LIN {X 0,Y 366.055,Z 486.683,A -85,B 0,C 180,E1 -21663.434,E2 -21663.434} C_VEL
LIN {X 0,Y 364.924,Z 500.957,A -85,B 0,C 180,E1 -21663.921,E2 -21663.921} C_VEL
LIN {X 0,Y 363.137,Z 514.776,A -85,B 0,C 180,E1 -21664.588,E2 -21664.588} C_VEL
LIN {X 0,Y 361.174,Z 526.804,A -85,B 0,C 180,E1 -21665.361,E2 -21665.361} C_VEL
LIN {X 0,Y 358.835,Z 539.501,A -85,B 0,C 180,E1 -21666.415,E2 -21666.415} C_VEL
LIN {X 0,Y 356.342,Z 551.532,A -85,B 0,C 180,E1 -21667.677,E2 -21667.677} C_VEL
LIN {X 0,Y 353.739,Z 562.686,A -85,B 0,C 180,E1 -21669.123,E2 -21669.123} C_VEL
LIN {X 0,Y 351.083,Z 573.104,A -85,B 0,C 180,E1 -21670.784,E2 -21670.784} C_VEL
LIN {X 0,Y 348.812,Z 581.735,A -85,B 0,C 180,E1 -21672.473,E2 -21672.473} C_VEL
LIN {X 0,Y 346.741,Z 590.061,A -85,B 0,C 180,E1 -21674.478,E2 -21674.478} C_VEL
LIN {X 0,Y 345.082,Z 596.796,A -85,B 0,C 180,E1 -21676.504,E2 -21676.504} C_VEL
LIN {X 0,Y 343.677,Z 602.83,A -85,B 0,C 180,E1 -21678.839,E2 -21678.839} C_VEL
LIN {X 0,Y 342.95,Z 606.345,A -85,B 0,C 180,E1 -21680.599,E2 -21680.599} C_VEL
LIN {X 0,Y 342.378,Z 609.772,A -85,B 0,C 180,E1 -21682.952,E2 -21682.952} C_VEL
LIN {X 0,Y 342.438,Z 612.217,A -85,B 0,C 180,E1 -21685.604,E2 -21685.604} C_VEL
LIN {X 0,Y 342.403,Z 616.736,A -85,B 0,C 180,E1 -21687.658,E2 -21687.658} C_VEL
LIN {X 0,Y 342.425,Z 618.738,A -85,B 0,C 180,E1 -21688.831,E2 -21688.831} C_VEL
LIN {X 0,Y 342.348,Z 621.565,A -85,B 0,C 180,E1 -21691.175,E2 -21691.175} C_VEL
LIN {X 0,Y 342.211,Z 622.906,A -85,B 0,C 180,E1 -21693.523,E2 -21693.523} C_VEL
LIN {X 0,Y 342.409,Z 622.824,A -85,B 0,C 180,E1 -21695.873,E2 -21695.873} C_VEL
LIN {X 0,Y 342.854,Z 621.327,A -85,B 0,C 180,E1 -21698.225,E2 -21698.225} C_VEL
LIN {X 0,Y 344.003,Z 618.414,A -85,B 0,C 180,E1 -21700.562,E2 -21700.562} C_VEL
LIN {X 0,Y 345.62,Z 614.037,A -85,B 0,C 180,E1 -21702.884,E2 -21702.884} C_VEL
LIN {X 0,Y 347.136,Z 609.753,A -85,B 0,C 180,E1 -21704.612,E2 -21704.612} C_VEL
LIN {X 0,Y 349.775,Z 602.476,A -85,B 0,C 180,E1 -21706.883,E2 -21706.883} C_VEL
LIN {X 0,Y 352.529,Z 594.517,A -85,B 0,C 180,E1 -21708.839,E2 -21708.839} C_VEL
LIN {X 0,Y 355.143,Z 586.331,A -85,B 0,C 180,E1 -21710.495,E2 -21710.495} C_VEL
LIN {X 0,Y 358.31,Z 576.517,A -85,B 0,C 180,E1 -21712.108,E2 -21712.108} C_VEL
LIN {X 0,Y 361.68,Z 564.796,A -85,B 0,C 180,E1 -21713.697,E2 -21713.697} C_VEL
LIN {X 0,Y 364.915,Z 552.862,A -85,B 0,C 180,E1 -21714.981,E2 -21714.981} C_VEL
LIN {X 0,Y 367.967,Z 539.899,A -85,B 0,C 180,E1 -21716.119,E2 -21716.119} C_VEL
LIN {X 0,Y 370.614,Z 527.481,A -85,B 0,C 180,E1 -21716.977,E2 -21716.977} C_VEL
LIN {X 0,Y 372.935,Z 514.221,A -85,B 0,C 180,E1 -21717.703,E2 -21717.703} C_VEL
LIN {X 0,Y 375.156,Z 498.538,A -85,B 0,C 180,E1 -21718.326,E2 -21718.326} C_VEL
LIN {X 0,Y 383.083,Z 416.624,A -85,B 0,C 180,E1 -21720.797,E2 -21720.797} C_VEL
LIN {X 0,Y 382.44,Z 396.943,A -85,B 0,C 180,E1 -21721.901,E2 -21721.901} C_VEL
LIN {X 0,Y 380.969,Z 378.673,A -85,B 0,C 180,E1 -21723.164,E2 -21723.164} C_VEL
LIN {X 0,Y 380.508,Z 375.676,A -85,B 0,C 180,E1 -21723.428,E2 -21723.428} C_VEL
LIN {X 0,Y 378.135,Z 368.085,A -85,B 0,C 180,E1 -21724.4,E2 -21724.4} C_VEL
LIN {X 0,Y 372.813,Z 359.888,A -85,B 0,C 180,E1 -21726.277,E2 -21726.277} C_VEL
LIN {X 0,Y 367.268,Z 352.213,A -85,B 0,C 180,E1 -21728.561,E2 -21728.561} C_VEL
LIN {X 0,Y 364.472,Z 347.395,A -85,B 0,C 180,E1 -21730.802,E2 -21730.802} C_VEL
LIN {X 0,Y 362.586,Z 344.058,A -85,B 0,C 180,E1 -21732.77,E2 -21732.77} C_VEL
LIN {X 0,Y 360.384,Z 340.995,A -85,B 0,C 180,E1 -21735.597,E2 -21735.597} C_VEL
LIN {X 0,Y 359.374,Z 339.035,A -85,B 0,C 180,E1 -21738.495,E2 -21738.495} C_VEL
LIN {X 0,Y 359.081,Z 338.68,A -85,B 0,C 180,E1 -21739.93,E2 -21739.93} C_VEL
LIN {X 0,Y 358.94,Z 338.821,A -85,B 0,C 180,E1 -21741.358,E2 -21741.358} C_VEL
LIN {X 0,Y 359.063,Z 340.127,A -85,B 0,C 180,E1 -21744.181,E2 -21744.181} C_VEL
LIN {X 0,Y 359.917,Z 342.545,A -85,B 0,C 180,E1 -21746.981,E2 -21746.981} C_VEL
LIN {X 0,Y 361.292,Z 346.17,A -85,B 0,C 180,E1 -21749.73,E2 -21749.73} C_VEL
LIN {X 0,Y 362.561,Z 349.811,A -85,B 0,C 180,E1 -21751.77,E2 -21751.77} C_VEL
LIN {X 0,Y 367.024,Z 356.698,A -85,B 0,C 180,E1 -21754.033,E2 -21754.033} C_VEL
LIN {X 0,Y 370.271,Z 361.948,A -85,B 0,C 180,E1 -21755.437,E2 -21755.437} C_VEL
LIN {X 0,Y 373.65,Z 367.876,A -85,B 0,C 180,E1 -21756.763,E2 -21756.763} C_VEL
LIN {X 0,Y 377.509,Z 375.052,A -85,B 0,C 180,E1 -21758.145,E2 -21758.145} C_VEL
LIN {X 0,Y 382.443,Z 385.972,A -85,B 0,C 180,E1 -21759.817,E2 -21759.817} C_VEL
LIN {X 0,Y 383.625,Z 389.184,A -85,B 0,C 180,E1 -21760.215,E2 -21760.215} C_VEL
LIN {X 0,Y 384.825,Z 399.873,A -85,B 0,C 180,E1 -21760.981,E2 -21760.981} C_VEL
LIN {X 0,Y 375.817,Z 490.766,A -85,B 0,C 180,E1 -21763.696,E2 -21763.696} C_VEL
LIN {X 0,Y 373.695,Z 505.863,A -85,B 0,C 180,E1 -21764.369,E2 -21764.369} C_VEL
LIN {X 0,Y 371.24,Z 520.286,A -85,B 0,C 180,E1 -21765.243,E2 -21765.243} C_VEL
LIN {X 0,Y 368.417,Z 533.693,A -85,B 0,C 180,E1 -21766.276,E2 -21766.276} C_VEL
LIN {X 0,Y 365.648,Z 545.087,A -85,B 0,C 180,E1 -21767.372,E2 -21767.372} C_VEL
LIN {X 0,Y 362.523,Z 556.587,A -85,B 0,C 180,E1 -21768.718,E2 -21768.718} C_VEL
LIN {X 0,Y 359.5,Z 566.8,A -85,B 0,C 180,E1 -21770.184,E2 -21770.184} C_VEL
LIN {X 0,Y 356.513,Z 576.165,A -85,B 0,C 180,E1 -21771.811,E2 -21771.811} C_VEL
LIN {X 0,Y 353.399,Z 585.186,A -85,B 0,C 180,E1 -21773.742,E2 -21773.742} C_VEL
LIN {X 0,Y 350.892,Z 591.603,A -85,B 0,C 180,E1 -21775.42,E2 -21775.42} C_VEL
LIN {X 0,Y 348.777,Z 596.889,A -85,B 0,C 180,E1 -21777.122,E2 -21777.122} C_VEL
LIN {X 0,Y 346.492,Z 602.436,A -85,B 0,C 180,E1 -21779.421,E2 -21779.421} C_VEL
LIN {X 0,Y 345.156,Z 605.533,A -85,B 0,C 180,E1 -21781.163,E2 -21781.163} C_VEL
LIN {X 0,Y 343.894,Z 608.425,A -85,B 0,C 180,E1 -21783.563,E2 -21783.563} C_VEL
LIN {X 0,Y 342.925,Z 609.815,A -85,B 0,C 180,E1 -21785.862,E2 -21785.862} C_VEL
LIN {X 0,Y 342.295,Z 609.846,A -85,B 0,C 180,E1 -21788.235,E2 -21788.235} C_VEL
LIN {X 0,Y 342.083,Z 608.426,A -85,B 0,C 180,E1 -21790.619,E2 -21790.619} C_VEL
LIN {X 0,Y 341.946,Z 605.459,A -85,B 0,C 180,E1 -21793.022,E2 -21793.022} C_VEL
LIN {X 0,Y 342.078,Z 602.213,A -85,B 0,C 180,E1 -21794.83,E2 -21794.83} C_VEL
LIN {X 0,Y 342.277,Z 597.919,A -85,B 0,C 180,E1 -21796.648,E2 -21796.648} C_VEL
LIN {X 0,Y 342.562,Z 591.515,A -85,B 0,C 180,E1 -21798.787,E2 -21798.787} C_VEL
LIN {X 0,Y 343.068,Z 583.313,A -85,B 0,C 180,E1 -21800.934,E2 -21800.934} C_VEL
LIN {X 0,Y 343.699,Z 573.569,A -85,B 0,C 180,E1 -21802.983,E2 -21802.983} C_VEL
LIN {X 0,Y 344.435,Z 563.987,A -85,B 0,C 180,E1 -21804.638,E2 -21804.638} C_VEL
LIN {X 0,Y 345.258,Z 553.252,A -85,B 0,C 180,E1 -21806.184,E2 -21806.184} C_VEL
LIN {X 0,Y 346.21,Z 541.181,A -85,B 0,C 180,E1 -21807.613,E2 -21807.613} C_VEL
LIN {X 0,Y 347.26,Z 527.207,A -85,B 0,C 180,E1 -21808.953,E2 -21808.953} C_VEL
LIN {X 0,Y 348.192,Z 513.062,A -85,B 0,C 180,E1 -21810.026,E2 -21810.026} C_VEL
LIN {X 0,Y 349.048,Z 498.453,A -85,B 0,C 180,E1 -21810.862,E2 -21810.862} C_VEL
LIN {X 0,Y 349.81,Z 482.818,A -85,B 0,C 180,E1 -21811.499,E2 -21811.499} C_VEL
LIN {X 0,Y 353.103,Z 383.38,A -85,B 0,C 180,E1 -21814.323,E2 -21814.323} C_VEL
LIN {X 0,Y 349.382,Z 350.073,A -85,B 0,C 180,E1 -21815.44,E2 -21815.44} C_VEL
LIN {X 0,Y 349.055,Z 345.645,A -85,B 0,C 180,E1 -21815.587,E2 -21815.587} C_VEL
LIN {X 0,Y 349.57,Z 337.879,A -85,B 0,C 180,E1 -21816.95,E2 -21816.95} C_VEL
LIN {X 0,Y 346.602,Z 322.549,A -85,B 0,C 180,E1 -21819.828,E2 -21819.828} C_VEL
LIN {X 0,Y 344.862,Z 314.085,A -85,B 0,C 180,E1 -21821.46,E2 -21821.46} C_VEL
LIN {X 0,Y 344.806,Z 314.085,A -85,B 0,C 180,E1 -21825.316,E2 -21825.316} C_VEL
LIN {X 0,Y 344.819,Z 314.088,A -85,B 0,C 180,E1 -21828.729,E2 -21828.729} C_VEL
LIN {X 0,Y 344.839,Z 314.089,A -85,B 0,C 180,E1 -21832.454,E2 -21832.454} C_VEL
LIN {X 0,Y 344.839,Z 314.08,A -85,B 0,C 180,E1 -21836.388,E2 -21836.388} C_VEL
LIN {X 0,Y 344.826,Z 314.088,A -85,B 0,C 180,E1 -21839.478,E2 -21839.478} C_VEL
LIN {X 0,Y 344.883,Z 314.078,A -85,B 0,C 180,E1 -21843.458,E2 -21843.458} C_VEL
LIN {X 0,Y 344.895,Z 314.079,A -85,B 0,C 180,E1 -21847.3,E2 -21847.3} C_VEL
LIN {X 0,Y 344.938,Z 314.077,A -85,B 0,C 180,E1 -21849.803,E2 -21849.803} C_VEL
LIN {X 0,Y 344.982,Z 314.067,A -85,B 0,C 180,E1 -21853.483,E2 -21853.483} C_VEL
LIN {X 0,Y 345.054,Z 314.156,A -85,B 0,C 180,E1 -21856.537,E2 -21856.537} C_VEL
LIN {X 0,Y 346.568,Z 318.213,A -85,B 0,C 180,E1 -21856.725,E2 -21856.725} C_VEL
LIN {X 0,Y 351.173,Z 329.859,A -85,B 0,C 180,E1 -21857.271,E2 -21857.271} C_VEL
LIN {X 0,Y 356.843,Z 346.888,A -85,B 0,C 180,E1 -21857.977,E2 -21857.977} C_VEL
LIN {X 0,Y 354.437,Z 447.995,A -85,B 0,C 180,E1 -21860.004,E2 -21860.004} C_VEL
LIN {X 0,Y 353.812,Z 462.506,A -85,B 0,C 180,E1 -21860.526,E2 -21860.526} C_VEL
LIN {X 0,Y 352.973,Z 476.914,A -85,B 0,C 180,E1 -21861.294,E2 -21861.294} C_VEL
LIN {X 0,Y 351.93,Z 488.862,A -85,B 0,C 180,E1 -21862.133,E2 -21862.133} C_VEL
LIN {X 0,Y 350.837,Z 500.065,A -85,B 0,C 180,E1 -21863.117,E2 -21863.117} C_VEL
LIN {X 0,Y 349.324,Z 511.865,A -85,B 0,C 180,E1 -21864.388,E2 -21864.388} C_VEL
LIN {X 0,Y 348.282,Z 521.61,A -85,B 0,C 180,E1 -21865.672,E2 -21865.672} C_VEL
LIN {X 0,Y 347.134,Z 530.782,A -85,B 0,C 180,E1 -21867.106,E2 -21867.106} C_VEL
LIN {X 0,Y 345.831,Z 539.993,A -85,B 0,C 180,E1 -21868.837,E2 -21868.837} C_VEL
LIN {X 0,Y 344.833,Z 547.662,A -85,B 0,C 180,E1 -21870.579,E2 -21870.579} C_VEL
LIN {X 0,Y 344.135,Z 554.022,A -85,B 0,C 180,E1 -21872.33,E2 -21872.33} C_VEL
LIN {X 0,Y 343.661,Z 559.279,A -85,B 0,C 180,E1 -21874.088,E2 -21874.088} C_VEL
LIN {X 0,Y 342.988,Z 564.867,A -85,B 0,C 180,E1 -21876.446,E2 -21876.446} C_VEL
LIN {X 0,Y 342.651,Z 568.004,A -85,B 0,C 180,E1 -21878.224,E2 -21878.224} C_VEL
LIN {X 0,Y 342.579,Z 570.938,A -85,B 0,C 180,E1 -21880.601,E2 -21880.601} C_VEL
LIN {X 0,Y 342.606,Z 572.515,A -85,B 0,C 180,E1 -21882.993,E2 -21882.993} C_VEL
LIN {X 0,Y 342.927,Z 572.738,A -85,B 0,C 180,E1 -21885.395,E2 -21885.395} C_VEL
LIN {X 0,Y 343.503,Z 571.602,A -85,B 0,C 180,E1 -21887.807,E2 -21887.807} C_VEL
LIN {X 0,Y 344.465,Z 569.036,A -85,B 0,C 180,E1 -21890.22,E2 -21890.22} C_VEL
LIN {X 0,Y 345.851,Z 564.953,A -85,B 0,C 180,E1 -21892.628,E2 -21892.628} C_VEL
LIN {X 0,Y 347.611,Z 559.233,A -85,B 0,C 180,E1 -21895.03,E2 -21895.03} C_VEL
LIN {X 0,Y 349.574,Z 552.707,A -85,B 0,C 180,E1 -21897.116,E2 -21897.116} C_VEL
LIN {X 0,Y 351.883,Z 544.776,A -85,B 0,C 180,E1 -21899.12,E2 -21899.12} C_VEL
LIN {X 0,Y 354.236,Z 535.872,A -85,B 0,C 180,E1 -21900.934,E2 -21900.934} C_VEL
LIN {X 0,Y 356.818,Z 525.291,A -85,B 0,C 180,E1 -21902.668,E2 -21902.668} C_VEL
LIN {X 0,Y 359.163,Z 514.547,A -85,B 0,C 180,E1 -21904.099,E2 -21904.099} C_VEL
LIN {X 0,Y 361.532,Z 502.269,A -85,B 0,C 180,E1 -21905.42,E2 -21905.42} C_VEL
LIN {X 0,Y 363.519,Z 489.69,A -85,B 0,C 180,E1 -21906.502,E2 -21906.502} C_VEL
LIN {X 0,Y 365.141,Z 475.959,A -85,B 0,C 180,E1 -21907.431,E2 -21907.431} C_VEL
LIN {X 0,Y 366.527,Z 461.755,A -85,B 0,C 180,E1 -21908.123,E2 -21908.123} C_VEL
LIN {X 0,Y 367.394,Z 447.635,A -85,B 0,C 180,E1 -21908.586,E2 -21908.586} C_VEL
LIN {X 0,Y 370.195,Z 363.744,A -85,B 0,C 180,E1 -21910.241,E2 -21910.241} C_VEL
LIN {X 0,Y 361.979,Z 345.819,A -85,B 0,C 180,E1 -21911.518,E2 -21911.518} C_VEL
LIN {X 0,Y 353.326,Z 329.446,A -85,B 0,C 180,E1 -21912.891,E2 -21912.891} C_VEL
LIN {X 0,Y 346.517,Z 317.849,A -85,B 0,C 180,E1 -21914.006,E2 -21914.006} C_VEL
LIN {X 0,Y 345.037,Z 315.104,A -85,B 0,C 180,E1 -21914.262,E2 -21914.262} C_VEL
LIN {X 0,Y 344.79,Z 314.078,A -85,B 0,C 180,E1 -21914.566,E2 -21914.566} C_VEL
LIN {X 0,Y 344.782,Z 314.085,A -85,B 0,C 180,E1 -21916.034,E2 -21916.034} C_VEL
LIN {X 0,Y 344.132,Z 314.178,A -85,B 0,C 180,E1 -21917.008,E2 -21917.008} C_VEL
LIN {X 0,Y 341.252,Z 314.534,A -85,B 0,C 180,E1 -21918.591,E2 -21918.591} C_VEL
LIN {X 0,Y 338.818,Z 314.835,A -85,B 0,C 180,E1 -21919.874,E2 -21919.874} C_VEL
LIN {X 0,Y 337.804,Z 314.962,A -85,B 0,C 180,E1 -21920.867,E2 -21920.867} C_VEL
LIN {X 0,Y 337.739,Z 314.971,A -85,B 0,C 180,E1 -21921.203,E2 -21921.203} C_VEL
LIN {X 0,Y 337.782,Z 314.932,A -85,B 0,C 180,E1 -21924.506,E2 -21924.506} C_VEL
LIN {X 0,Y 337.796,Z 314.961,A -85,B 0,C 180,E1 -21928.223,E2 -21928.223} C_VEL
LIN {X 0,Y 337.823,Z 314.959,A -85,B 0,C 180,E1 -21931.518,E2 -21931.518} C_VEL
LIN {X 0,Y 337.82,Z 314.957,A -85,B 0,C 180,E1 -21935.501,E2 -21935.501} C_VEL
LIN {X 0,Y 337.877,Z 314.955,A -85,B 0,C 180,E1 -21939.364,E2 -21939.364} C_VEL
LIN {X 0,Y 337.892,Z 314.952,A -85,B 0,C 180,E1 -21943.129,E2 -21943.129} C_VEL
LIN {X 0,Y 338.007,Z 314.927,A -85,B 0,C 180,E1 -21946.882,E2 -21946.882} C_VEL
LIN {X 0,Y 338.028,Z 314.921,A -85,B 0,C 180,E1 -21950.458,E2 -21950.458} C_VEL
LIN {X 0,Y 338.186,Z 314.916,A -85,B 0,C 180,E1 -21954.056,E2 -21954.056} C_VEL
LIN {X 0,Y 338.218,Z 314.902,A -85,B 0,C 180,E1 -21957.626,E2 -21957.626} C_VEL
LIN {X 0,Y 338.191,Z 314.898,A -85,B 0,C 180,E1 -21961.187,E2 -21961.187} C_VEL
LIN {X 0,Y 338.226,Z 314.913,A -85,B 0,C 180,E1 -21964.752,E2 -21964.752} C_VEL
LIN {X 0,Y 338.075,Z 314.915,A -85,B 0,C 180,E1 -21968.339,E2 -21968.339} C_VEL
LIN {X 0,Y 338.021,Z 314.919,A -85,B 0,C 180,E1 -21971.959,E2 -21971.959} C_VEL
LIN {X 0,Y 337.911,Z 314.945,A -85,B 0,C 180,E1 -21975.633,E2 -21975.633} C_VEL
LIN {X 0,Y 337.863,Z 314.939,A -85,B 0,C 180,E1 -21978.118,E2 -21978.118} C_VEL
LIN {X 0,Y 337.863,Z 314.947,A -85,B 0,C 180,E1 -21981.115,E2 -21981.115} C_VEL
LIN {X 0,Y 337.82,Z 314.964,A -85,B 0,C 180,E1 -21984.5,E2 -21984.5} C_VEL
LIN {X 0,Y 337.823,Z 314.964,A -85,B 0,C 180,E1 -21988.482,E2 -21988.482} C_VEL
LIN {X 0,Y 337.801,Z 314.962,A -85,B 0,C 180,E1 -21991.779,E2 -21991.779} C_VEL
LIN {X 0,Y 337.829,Z 314.92,A -85,B 0,C 180,E1 -21995.489,E2 -21995.489} C_VEL
LIN {X 0,Y 337.832,Z 314.959,A -85,B 0,C 180,E1 -21998.463,E2 -21998.463} C_VEL
LIN {X 0,Y 337.803,Z 314.966,A -85,B 0,C 180,E1 -22001.72,E2 -22001.72} C_VEL
LIN {X 0,Y 337.796,Z 314.96,A -85,B 0,C 180,E1 -22005.174,E2 -22005.174} C_VEL
LIN {X 0,Y 337.835,Z 314.994,A -85,B 0,C 180,E1 -22008.144,E2 -22008.144} C_VEL
LIN {X 0,Y 341.432,Z 327.545,A -85,B 0,C 180,E1 -22012.321,E2 -22012.321} C_VEL
LIN {X 0,Y 344.132,Z 338.395,A -85,B 0,C 180,E1 -22015.595,E2 -22015.595} C_VEL
LIN {X 0,Y 345.966,Z 346.803,A -85,B 0,C 180,E1 -22017.913,E2 -22017.913} C_VEL
LIN {X 0,Y 354.721,Z 365.775,A -85,B 0,C 180,E1 -22019.409,E2 -22019.409} C_VEL
LIN {X 0,Y 360.3,Z 397.531,A -85,B 0,C 180,E1 -22020.776,E2 -22020.776} C_VEL
LIN {X 0,Y 362.564,Z 414.669,A -85,B 0,C 180,E1 -22021.409,E2 -22021.409} C_VEL
LIN {X 0,Y 360.53,Z 473.255,A -85,B 0,C 180,E1 -22022.564,E2 -22022.564} C_VEL
LIN {X 0,Y 359.715,Z 490.214,A -85,B 0,C 180,E1 -22022.967,E2 -22022.967} C_VEL
LIN {X 0,Y 358.306,Z 504.713,A -85,B 0,C 180,E1 -22023.519,E2 -22023.519} C_VEL
LIN {X 0,Y 356.373,Z 518.008,A -85,B 0,C 180,E1 -22024.227,E2 -22024.227} C_VEL
LIN {X 0,Y 354.175,Z 530.938,A -85,B 0,C 180,E1 -22025.153,E2 -22025.153} C_VEL
LIN {X 0,Y 351.494,Z 544.041,A -85,B 0,C 180,E1 -22026.36,E2 -22026.36} C_VEL
LIN {X 0,Y 348.884,Z 555.826,A -85,B 0,C 180,E1 -22027.735,E2 -22027.735} C_VEL
LIN {X 0,Y 346.211,Z 566.513,A -85,B 0,C 180,E1 -22029.268,E2 -22029.268} C_VEL
LIN {X 0,Y 343.558,Z 576.181,A -85,B 0,C 180,E1 -22030.965,E2 -22030.965} C_VEL
LIN {X 0,Y 341.389,Z 584.236,A -85,B 0,C 180,E1 -22032.696,E2 -22032.696} C_VEL
LIN {X 0,Y 339.34,Z 591.996,A -85,B 0,C 180,E1 -22034.745,E2 -22034.745} C_VEL
LIN {X 0,Y 337.72,Z 598.264,A -85,B 0,C 180,E1 -22036.815,E2 -22036.815} C_VEL
LIN {X 0,Y 336.364,Z 603.864,A -85,B 0,C 180,E1 -22039.201,E2 -22039.201} C_VEL
LIN {X 0,Y 335.534,Z 607.949,A -85,B 0,C 180,E1 -22041.6,E2 -22041.6} C_VEL
LIN {X 0,Y 335.275,Z 610.63,A -85,B 0,C 180,E1 -22044.007,E2 -22044.007} C_VEL
LIN {X 0,Y 335.369,Z 611.745,A -85,B 0,C 180,E1 -22045.661,E2 -22045.661} C_VEL
LIN {X 0,Y 335.337,Z 616.072,A -85,B 0,C 180,E1 -22047.609,E2 -22047.609} C_VEL
LIN {X 0,Y 335.361,Z 618.154,A -85,B 0,C 180,E1 -22048.806,E2 -22048.806} C_VEL
LIN {X 0,Y 335.259,Z 621.129,A -85,B 0,C 180,E1 -22051.2,E2 -22051.2} C_VEL
LIN {X 0,Y 335.135,Z 622.628,A -85,B 0,C 180,E1 -22053.598,E2 -22053.598} C_VEL
LIN {X 0,Y 335.333,Z 622.712,A -85,B 0,C 180,E1 -22055.998,E2 -22055.998} C_VEL
LIN {X 0,Y 335.815,Z 621.404,A -85,B 0,C 180,E1 -22058.398,E2 -22058.398} C_VEL
LIN {X 0,Y 337.027,Z 618.708,A -85,B 0,C 180,E1 -22060.783,E2 -22060.783} C_VEL
LIN {X 0,Y 338.709,Z 614.527,A -85,B 0,C 180,E1 -22063.151,E2 -22063.151} C_VEL
LIN {X 0,Y 340.3,Z 610.395,A -85,B 0,C 180,E1 -22064.912,E2 -22064.912} C_VEL
LIN {X 0,Y 342.289,Z 605.295,A -85,B 0,C 180,E1 -22066.651,E2 -22066.651} C_VEL
LIN {X 0,Y 345.123,Z 598.05,A -85,B 0,C 180,E1 -22068.645,E2 -22068.645} C_VEL
LIN {X 0,Y 348.18,Z 589.205,A -85,B 0,C 180,E1 -22070.616,E2 -22070.616} C_VEL
LIN {X 0,Y 351.359,Z 580.05,A -85,B 0,C 180,E1 -22072.26,E2 -22072.26} C_VEL
LIN {X 0,Y 354.814,Z 569.048,A -85,B 0,C 180,E1 -22073.875,E2 -22073.875} C_VEL
LIN {X 0,Y 358.024,Z 558.119,A -85,B 0,C 180,E1 -22075.186,E2 -22075.186} C_VEL
LIN {X 0,Y 361.492,Z 544.897,A -85,B 0,C 180,E1 -22076.468,E2 -22076.468} C_VEL
LIN {X 0,Y 364.49,Z 531.947,A -85,B 0,C 180,E1 -22077.468,E2 -22077.468} C_VEL
LIN {X 0,Y 367.359,Z 517.613,A -85,B 0,C 180,E1 -22078.316,E2 -22078.316} C_VEL
LIN {X 0,Y 369.846,Z 501.857,A -85,B 0,C 180,E1 -22078.996,E2 -22078.996} C_VEL
LIN {X 0,Y 374.454,Z 456.543,A -85,B 0,C 180,E1 -22080.414,E2 -22080.414} C_VEL
LIN {X 0,Y 378.481,Z 416.881,A -85,B 0,C 180,E1 -22081.645,E2 -22081.645} C_VEL
LIN {X 0,Y 377.992,Z 398.003,A -85,B 0,C 180,E1 -22082.745,E2 -22082.745} C_VEL
LIN {X 0,Y 376.744,Z 380.772,A -85,B 0,C 180,E1 -22083.984,E2 -22083.984} C_VEL
LIN {X 0,Y 374.639,Z 373.203,A -85,B 0,C 180,E1 -22084.941,E2 -22084.941} C_VEL
LIN {X 0,Y 369.188,Z 364.748,A -85,B 0,C 180,E1 -22086.976,E2 -22086.976} C_VEL
LIN {X 0,Y 364.06,Z 357.643,A -85,B 0,C 180,E1 -22089.224,E2 -22089.224} C_VEL
LIN {X 0,Y 359.593,Z 351.887,A -85,B 0,C 180,E1 -22091.649,E2 -22091.649} C_VEL
LIN {X 0,Y 357.856,Z 348.927,A -85,B 0,C 180,E1 -22093.596,E2 -22093.596} C_VEL
LIN {X 0,Y 355.846,Z 345.925,A -85,B 0,C 180,E1 -22096.747,E2 -22096.747} C_VEL
LIN {X 0,Y 355.274,Z 344.83,A -85,B 0,C 180,E1 -22098.524,E2 -22098.524} C_VEL
LIN {X 0,Y 354.812,Z 344.484,A -85,B 0,C 180,E1 -22100.823,E2 -22100.823} C_VEL
LIN {X 0,Y 354.708,Z 345.503,A -85,B 0,C 180,E1 -22103.672,E2 -22103.672} C_VEL
LIN {X 0,Y 355.349,Z 347.627,A -85,B 0,C 180,E1 -22106.501,E2 -22106.501} C_VEL
LIN {X 0,Y 356.369,Z 350.397,A -85,B 0,C 180,E1 -22108.753,E2 -22108.753} C_VEL
LIN {X 0,Y 360.406,Z 356.353,A -85,B 0,C 180,E1 -22111.501,E2 -22111.501} C_VEL
LIN {X 0,Y 364.515,Z 362.972,A -85,B 0,C 180,E1 -22113.681,E2 -22113.681} C_VEL
LIN {X 0,Y 367.502,Z 367.96,A -85,B 0,C 180,E1 -22115.035,E2 -22115.035} C_VEL
LIN {X 0,Y 370.33,Z 373.094,A -85,B 0,C 180,E1 -22116.214,E2 -22116.214} C_VEL
LIN {X 0,Y 374.096,Z 380.396,A -85,B 0,C 180,E1 -22117.655,E2 -22117.655} C_VEL
LIN {X 0,Y 378.778,Z 391.171,A -85,B 0,C 180,E1 -22119.331,E2 -22119.331} C_VEL
LIN {X 0,Y 379.528,Z 393.855,A -85,B 0,C 180,E1 -22119.633,E2 -22119.633} C_VEL
LIN {X 0,Y 380.267,Z 401.987,A -85,B 0,C 180,E1 -22120.21,E2 -22120.21} C_VEL
LIN {X 0,Y 370.923,Z 491.049,A -85,B 0,C 180,E1 -22122.91,E2 -22122.91} C_VEL
LIN {X 0,Y 368.51,Z 507.23,A -85,B 0,C 180,E1 -22123.647,E2 -22123.647} C_VEL
LIN {X 0,Y 365.77,Z 522.26,A -85,B 0,C 180,E1 -22124.591,E2 -22124.591} C_VEL
LIN {X 0,Y 362.807,Z 535.253,A -85,B 0,C 180,E1 -22125.637,E2 -22125.637} C_VEL
LIN {X 0,Y 359.616,Z 547.652,A -85,B 0,C 180,E1 -22126.883,E2 -22126.883} C_VEL
LIN {X 0,Y 356.678,Z 557.669,A -85,B 0,C 180,E1 -22128.1,E2 -22128.1} C_VEL
LIN {X 0,Y 353.25,Z 568.582,A -85,B 0,C 180,E1 -22129.72,E2 -22129.72} C_VEL
LIN {X 0,Y 350.126,Z 577.673,A -85,B 0,C 180,E1 -22131.371,E2 -22131.371} C_VEL
LIN {X 0,Y 346.886,Z 586.436,A -85,B 0,C 180,E1 -22133.333,E2 -22133.333} C_VEL
LIN {X 0,Y 343.887,Z 593.578,A -85,B 0,C 180,E1 -22135.327,E2 -22135.327} C_VEL
LIN {X 0,Y 341.751,Z 598.563,A -85,B 0,C 180,E1 -22137.063,E2 -22137.063} C_VEL
LIN {X 0,Y 339.38,Z 603.688,A -85,B 0,C 180,E1 -22139.409,E2 -22139.409} C_VEL
LIN {X 0,Y 338.045,Z 606.533,A -85,B 0,C 180,E1 -22141.187,E2 -22141.187} C_VEL
LIN {X 0,Y 336.793,Z 609.036,A -85,B 0,C 180,E1 -22143.577,E2 -22143.577} C_VEL
LIN {X 0,Y 335.78,Z 610.13,A -85,B 0,C 180,E1 -22145.987,E2 -22145.987} C_VEL
LIN {X 0,Y 335.176,Z 609.808,A -85,B 0,C 180,E1 -22148.412,E2 -22148.412} C_VEL
LIN {X 0,Y 334.961,Z 608.044,A -85,B 0,C 180,E1 -22150.848,E2 -22150.848} C_VEL
LIN {X 0,Y 334.865,Z 604.762,A -85,B 0,C 180,E1 -22153.302,E2 -22153.302} C_VEL
LIN {X 0,Y 335.029,Z 601.207,A -85,B 0,C 180,E1 -22155.149,E2 -22155.149} C_VEL
LIN {X 0,Y 335.226,Z 596.631,A -85,B 0,C 180,E1 -22157.009,E2 -22157.009} C_VEL
LIN {X 0,Y 335.56,Z 589.792,A -85,B 0,C 180,E1 -22159.194,E2 -22159.194} C_VEL
LIN {X 0,Y 336.019,Z 582.49,A -85,B 0,C 180,E1 -22161.075,E2 -22161.075} C_VEL
LIN {X 0,Y 336.608,Z 573.584,A -85,B 0,C 180,E1 -22162.965,E2 -22162.965} C_VEL
LIN {X 0,Y 337.455,Z 562.728,A -85,B 0,C 180,E1 -22164.855,E2 -22164.855} C_VEL
LIN {X 0,Y 338.412,Z 550.451,A -85,B 0,C 180,E1 -22166.589,E2 -22166.589} C_VEL
LIN {X 0,Y 339.407,Z 538.043,A -85,B 0,C 180,E1 -22168.023,E2 -22168.023} C_VEL
LIN {X 0,Y 340.401,Z 524.846,A -85,B 0,C 180,E1 -22169.255,E2 -22169.255} C_VEL
LIN {X 0,Y 341.294,Z 510.254,A -85,B 0,C 180,E1 -22170.324,E2 -22170.324} C_VEL
LIN {X 0,Y 342.164,Z 494.994,A -85,B 0,C 180,E1 -22171.167,E2 -22171.167} C_VEL
LIN {X 0,Y 342.859,Z 479.942,A -85,B 0,C 180,E1 -22171.74,E2 -22171.74} C_VEL
LIN {X 0,Y 346.065,Z 383.456,A -85,B 0,C 180,E1 -22174.553,E2 -22174.553} C_VEL
LIN {X 0,Y 342.444,Z 350.529,A -85,B 0,C 180,E1 -22175.68,E2 -22175.68} C_VEL
LIN {X 0,Y 342.102,Z 345.671,A -85,B 0,C 180,E1 -22175.861,E2 -22175.861} C_VEL
LIN {X 0,Y 342.541,Z 338.645,A -85,B 0,C 180,E1 -22177.105,E2 -22177.105} C_VEL
LIN {X 0,Y 339.341,Z 322.415,A -85,B 0,C 180,E1 -22180.203,E2 -22180.203} C_VEL
LIN {X 0,Y 337.827,Z 314.962,A -85,B 0,C 180,E1 -22181.665,E2 -22181.665} C_VEL
LIN {X 0,Y 337.758,Z 314.963,A -85,B 0,C 180,E1 -22185.16,E2 -22185.16} C_VEL
LIN {X 0,Y 337.768,Z 314.97,A -85,B 0,C 180,E1 -22188.422,E2 -22188.422} C_VEL
LIN {X 0,Y 337.784,Z 314.967,A -85,B 0,C 180,E1 -22191.998,E2 -22191.998} C_VEL
LIN {X 0,Y 337.774,Z 314.961,A -85,B 0,C 180,E1 -22194.502,E2 -22194.502} C_VEL
LIN {X 0,Y 337.75,Z 314.964,A -85,B 0,C 180,E1 -22197.368,E2 -22197.368} C_VEL
LIN {X 0,Y 337.8,Z 314.96,A -85,B 0,C 180,E1 -22201.513,E2 -22201.513} C_VEL
LIN {X 0,Y 337.826,Z 314.964,A -85,B 0,C 180,E1 -22204.186,E2 -22204.186} C_VEL
LIN {X 0,Y 337.832,Z 314.959,A -85,B 0,C 180,E1 -22206.798,E2 -22206.798} C_VEL
LIN {X 0,Y 337.904,Z 314.951,A -85,B 0,C 180,E1 -22209.363,E2 -22209.363} C_VEL
LIN {X 0,Y 337.94,Z 314.943,A -85,B 0,C 180,E1 -22213.129,E2 -22213.129} C_VEL
LIN {X 0,Y 337.967,Z 314.946,A -85,B 0,C 180,E1 -22216.075,E2 -22216.075} C_VEL
LIN {X 0,Y 339.918,Z 320.014,A -85,B 0,C 180,E1 -22216.328,E2 -22216.328} C_VEL
LIN {X 0,Y 344.585,Z 331.537,A -85,B 0,C 180,E1 -22216.89,E2 -22216.89} C_VEL
LIN {X 0,Y 350.08,Z 347.995,A -85,B 0,C 180,E1 -22217.595,E2 -22217.595} C_VEL
LIN {X 0,Y 347.695,Z 448.719,A -85,B 0,C 180,E1 -22219.661,E2 -22219.661} C_VEL
LIN {X 0,Y 347.048,Z 463.122,A -85,B 0,C 180,E1 -22220.192,E2 -22220.192} C_VEL
LIN {X 0,Y 346.183,Z 477.476,A -85,B 0,C 180,E1 -22220.976,E2 -22220.976} C_VEL
LIN {X 0,Y 345.11,Z 489.393,A -85,B 0,C 180,E1 -22221.829,E2 -22221.829} C_VEL
LIN {X 0,Y 343.965,Z 500.581,A -85,B 0,C 180,E1 -22222.832,E2 -22222.832} C_VEL
LIN {X 0,Y 342.429,Z 512.362,A -85,B 0,C 180,E1 -22224.127,E2 -22224.127} C_VEL
LIN {X 0,Y 341.266,Z 523.056,A -85,B 0,C 180,E1 -22225.583,E2 -22225.583} C_VEL
LIN {X 0,Y 340.016,Z 532.074,A -85,B 0,C 180,E1 -22227.045,E2 -22227.045} C_VEL
LIN {X 0,Y 338.757,Z 541.13,A -85,B 0,C 180,E1 -22228.812,E2 -22228.812} C_VEL
LIN {X 0,Y 337.68,Z 548.685,A -85,B 0,C 180,E1 -22230.591,E2 -22230.591} C_VEL
LIN {X 0,Y 337.067,Z 554.964,A -85,B 0,C 180,E1 -22232.379,E2 -22232.379} C_VEL
LIN {X 0,Y 336.549,Z 560.131,A -85,B 0,C 180,E1 -22234.174,E2 -22234.174} C_VEL
LIN {X 0,Y 336.028,Z 564.368,A -85,B 0,C 180,E1 -22235.979,E2 -22235.979} C_VEL
LIN {X 0,Y 335.559,Z 568.664,A -85,B 0,C 180,E1 -22238.399,E2 -22238.399} C_VEL
LIN {X 0,Y 335.483,Z 571.512,A -85,B 0,C 180,E1 -22240.828,E2 -22240.828} C_VEL
LIN {X 0,Y 335.543,Z 573.002,A -85,B 0,C 180,E1 -22243.272,E2 -22243.272} C_VEL
LIN {X 0,Y 335.9,Z 573.137,A -85,B 0,C 180,E1 -22245.726,E2 -22245.726} C_VEL
LIN {X 0,Y 336.538,Z 571.889,A -85,B 0,C 180,E1 -22248.188,E2 -22248.188} C_VEL
LIN {X 0,Y 337.586,Z 569.215,A -85,B 0,C 180,E1 -22250.651,E2 -22250.651} C_VEL
LIN {X 0,Y 339.076,Z 565.036,A -85,B 0,C 180,E1 -22253.106,E2 -22253.106} C_VEL
LIN {X 0,Y 340.646,Z 560.13,A -85,B 0,C 180,E1 -22255.212,E2 -22255.212} C_VEL
LIN {X 0,Y 342.726,Z 553.599,A -85,B 0,C 180,E1 -22257.373,E2 -22257.373} C_VEL
LIN {X 0,Y 345.176,Z 545.525,A -85,B 0,C 180,E1 -22259.474,E2 -22259.474} C_VEL
LIN {X 0,Y 347.519,Z 536.998,A -85,B 0,C 180,E1 -22261.262,E2 -22261.262} C_VEL
LIN {X 0,Y 350.195,Z 526.631,A -85,B 0,C 180,E1 -22263.024,E2 -22263.024} C_VEL
LIN {X 0,Y 352.579,Z 516.079,A -85,B 0,C 180,E1 -22264.481,E2 -22264.481} C_VEL
LIN {X 0,Y 355.085,Z 503.805,A -85,B 0,C 180,E1 -22265.843,E2 -22265.843} C_VEL
LIN {X 0,Y 357.088,Z 491.798,A -85,B 0,C 180,E1 -22266.918,E2 -22266.918} C_VEL
LIN {X 0,Y 358.786,Z 478.552,A -85,B 0,C 180,E1 -22267.856,E2 -22267.856} C_VEL
LIN {X 0,Y 360.205,Z 464.962,A -85,B 0,C 180,E1 -22268.57,E2 -22268.57} C_VEL
LIN {X 0,Y 361.136,Z 451.762,A -85,B 0,C 180,E1 -22269.059,E2 -22269.059} C_VEL
LIN {X 0,Y 361.955,Z 428.744,A -85,B 0,C 180,E1 -22269.573,E2 -22269.573} C_VEL
LIN {X 0,Y 364.298,Z 366.01,A -85,B 0,C 180,E1 -22270.793,E2 -22270.793} C_VEL
LIN {X 0,Y 355.899,Z 347.799,A -85,B 0,C 180,E1 -22272.145,E2 -22272.145} C_VEL
LIN {X 0,Y 346.953,Z 331.003,A -85,B 0,C 180,E1 -22273.616,E2 -22273.616} C_VEL
LIN {X 0,Y 341.655,Z 322.217,A -85,B 0,C 180,E1 -22274.51,E2 -22274.51} C_VEL
LIN {X 0,Y 339.739,Z 319.047,A -85,B 0,C 180,E1 -22274.844,E2 -22274.844} C_VEL
LIN {X 0,Y 338.165,Z 316.591,A -85,B 0,C 180,E1 -22275.118,E2 -22275.118} C_VEL
LIN {X 0,Y 337.784,Z 315.189,A -85,B 0,C 180,E1 -22275.26,E2 -22275.26} C_VEL
LIN {X 0,Y 337.746,Z 314.956,A -85,B 0,C 180,E1 -22275.532,E2 -22275.532} C_VEL
LIN {X 0,Y 337.767,Z 314.967,A -85,B 0,C 180,E1 -22278.425,E2 -22278.425} C_VEL
LIN {X 0,Y 337.739,Z 314.971,A -85,B 0,C 180,E1 -22281.203,E2 -22281.203} C_VEL
LIN {X 0,Y 337.113,Z 315.051,A -85,B 0,C 180,E1 -22282.198,E2 -22282.198} C_VEL
LIN {X 0,Y 334.258,Z 315.392,A -85,B 0,C 180,E1 -22283.816,E2 -22283.816} C_VEL
LIN {X 0,Y 331.826,Z 315.685,A -85,B 0,C 180,E1 -22285.126,E2 -22285.126} C_VEL
LIN {X 0,Y 330.8,Z 315.82,A -85,B 0,C 180,E1 -22286.141,E2 -22286.141} C_VEL
LIN {X 0,Y 330.728,Z 315.836,A -85,B 0,C 180,E1 -22286.485,E2 -22286.485} C_VEL
LIN {X 0,Y 330.749,Z 315.841,A -85,B 0,C 180,E1 -22290.251,E2 -22290.251} C_VEL
LIN {X 0,Y 330.747,Z 315.835,A -85,B 0,C 180,E1 -22293.594,E2 -22293.594} C_VEL
LIN {X 0,Y 330.771,Z 315.828,A -85,B 0,C 180,E1 -22296.275,E2 -22296.275} C_VEL
LIN {X 0,Y 330.832,Z 315.833,A -85,B 0,C 180,E1 -22298.904,E2 -22298.904} C_VEL
LIN {X 0,Y 330.852,Z 315.827,A -85,B 0,C 180,E1 -22302.759,E2 -22302.759} C_VEL
LIN {X 0,Y 330.957,Z 315.804,A -85,B 0,C 180,E1 -22306.777,E2 -22306.777} C_VEL
LIN {X 0,Y 330.974,Z 315.801,A -85,B 0,C 180,E1 -22310.253,E2 -22310.253} C_VEL
LIN {X 0,Y 331.172,Z 315.79,A -85,B 0,C 180,E1 -22313.93,E2 -22313.93} C_VEL
LIN {X 0,Y 331.183,Z 315.777,A -85,B 0,C 180,E1 -22317.576,E2 -22317.576} C_VEL
LIN {X 0,Y 331.168,Z 315.772,A -85,B 0,C 180,E1 -22321.212,E2 -22321.212} C_VEL
LIN {X 0,Y 331.171,Z 315.792,A -85,B 0,C 180,E1 -22324.853,E2 -22324.853} C_VEL
LIN {X 0,Y 331.09,Z 315.779,A -85,B 0,C 180,E1 -22327.293,E2 -22327.293} C_VEL
LIN {X 0,Y 330.95,Z 315.808,A -85,B 0,C 180,E1 -22330.981,E2 -22330.981} C_VEL
LIN {X 0,Y 330.958,Z 315.8,A -85,B 0,C 180,E1 -22333.462,E2 -22333.462} C_VEL
LIN {X 0,Y 330.848,Z 315.81,A -85,B 0,C 180,E1 -22337.705,E2 -22337.705} C_VEL
LIN {X 0,Y 330.803,Z 315.824,A -85,B 0,C 180,E1 -22341.316,E2 -22341.316} C_VEL
LIN {X 0,Y 330.772,Z 315.837,A -85,B 0,C 180,E1 -22345.057,E2 -22345.057} C_VEL
LIN {X 0,Y 330.759,Z 315.839,A -85,B 0,C 180,E1 -22347.768,E2 -22347.768} C_VEL
LIN {X 0,Y 330.734,Z 315.835,A -85,B 0,C 180,E1 -22350.55,E2 -22350.55} C_VEL
LIN {X 0,Y 330.77,Z 315.81,A -85,B 0,C 180,E1 -22354.33,E2 -22354.33} C_VEL
LIN {X 0,Y 330.799,Z 315.824,A -85,B 0,C 180,E1 -22357.883,E2 -22357.883} C_VEL
LIN {X 0,Y 330.739,Z 315.842,A -85,B 0,C 180,E1 -22361.035,E2 -22361.035} C_VEL
LIN {X 0,Y 330.741,Z 315.844,A -85,B 0,C 180,E1 -22364.337,E2 -22364.337} C_VEL
LIN {X 0,Y 330.755,Z 315.92,A -85,B 0,C 180,E1 -22367.292,E2 -22367.292} C_VEL
LIN {X 0,Y 333.829,Z 326.37,A -85,B 0,C 180,E1 -22370.927,E2 -22370.927} C_VEL
LIN {X 0,Y 336.319,Z 335.836,A -85,B 0,C 180,E1 -22373.965,E2 -22373.965} C_VEL
LIN {X 0,Y 338.719,Z 346.188,A -85,B 0,C 180,E1 -22376.989,E2 -22376.989} C_VEL
LIN {X 0,Y 348.636,Z 367.385,A -85,B 0,C 180,E1 -22378.751,E2 -22378.751} C_VEL
LIN {X 0,Y 349.621,Z 370.849,A -85,B 0,C 180,E1 -22378.952,E2 -22378.952} C_VEL
LIN {X 0,Y 354.635,Z 400.615,A -85,B 0,C 180,E1 -22380.244,E2 -22380.244} C_VEL
LIN {X 0,Y 356.595,Z 415.78,A -85,B 0,C 180,E1 -22380.818,E2 -22380.818} C_VEL
LIN {X 0,Y 354.074,Z 484.709,A -85,B 0,C 180,E1 -22382.221,E2 -22382.221} C_VEL
LIN {X 0,Y 352.838,Z 499.406,A -85,B 0,C 180,E1 -22382.716,E2 -22382.716} C_VEL
LIN {X 0,Y 350.984,Z 513.402,A -85,B 0,C 180,E1 -22383.403,E2 -22383.403} C_VEL
LIN {X 0,Y 349.021,Z 524.674,A -85,B 0,C 180,E1 -22384.123,E2 -22384.123} C_VEL
LIN {X 0,Y 346.543,Z 537.618,A -85,B 0,C 180,E1 -22385.206,E2 -22385.206} C_VEL
LIN {X 0,Y 343.801,Z 549.885,A -85,B 0,C 180,E1 -22386.505,E2 -22386.505} C_VEL
LIN {X 0,Y 341.038,Z 561.131,A -85,B 0,C 180,E1 -22387.99,E2 -22387.99} C_VEL
LIN {X 0,Y 338.134,Z 571.668,A -85,B 0,C 180,E1 -22389.701,E2 -22389.701} C_VEL
LIN {X 0,Y 335.665,Z 580.396,A -85,B 0,C 180,E1 -22391.448,E2 -22391.448} C_VEL
LIN {X 0,Y 333.294,Z 588.811,A -85,B 0,C 180,E1 -22393.521,E2 -22393.521} C_VEL
LIN {X 0,Y 331.681,Z 594.714,A -85,B 0,C 180,E1 -22395.324,E2 -22395.324} C_VEL
LIN {X 0,Y 329.981,Z 601.068,A -85,B 0,C 180,E1 -22397.748,E2 -22397.748} C_VEL
LIN {X 0,Y 328.849,Z 605.833,A -85,B 0,C 180,E1 -22400.192,E2 -22400.192} C_VEL
LIN {X 0,Y 328.218,Z 609.133,A -85,B 0,C 180,E1 -22402.646,E2 -22402.646} C_VEL
LIN {X 0,Y 328.232,Z 611.09,A -85,B 0,C 180,E1 -22405.106,E2 -22405.106} C_VEL
LIN {X 0,Y 328.288,Z 611.62,A -85,B 0,C 180,E1 -22405.874,E2 -22405.874} C_VEL
LIN {X 0,Y 328.274,Z 616.469,A -85,B 0,C 180,E1 -22408.169,E2 -22408.169} C_VEL
LIN {X 0,Y 328.227,Z 619.308,A -85,B 0,C 180,E1 -22410.003,E2 -22410.003} C_VEL
LIN {X 0,Y 328.174,Z 620.687,A -85,B 0,C 180,E1 -22411.226,E2 -22411.226} C_VEL
LIN {X 0,Y 328.068,Z 622.343,A -85,B 0,C 180,E1 -22413.675,E2 -22413.675} C_VEL
LIN {X 0,Y 328.267,Z 622.593,A -85,B 0,C 180,E1 -22416.127,E2 -22416.127} C_VEL
LIN {X 0,Y 328.786,Z 621.461,A -85,B 0,C 180,E1 -22418.579,E2 -22418.579} C_VEL
LIN {X 0,Y 330.041,Z 618.942,A -85,B 0,C 180,E1 -22421.014,E2 -22421.014} C_VEL
LIN {X 0,Y 331.812,Z 615.004,A -85,B 0,C 180,E1 -22423.43,E2 -22423.43} C_VEL
LIN {X 0,Y 333.479,Z 611.023,A -85,B 0,C 180,E1 -22425.224,E2 -22425.224} C_VEL
LIN {X 0,Y 336.353,Z 604.304,A -85,B 0,C 180,E1 -22427.578,E2 -22427.578} C_VEL
LIN {X 0,Y 339.321,Z 596.911,A -85,B 0,C 180,E1 -22429.602,E2 -22429.602} C_VEL
LIN {X 0,Y 342.689,Z 587.854,A -85,B 0,C 180,E1 -22431.59,E2 -22431.59} C_VEL
LIN {X 0,Y 346.107,Z 578.474,A -85,B 0,C 180,E1 -22433.246,E2 -22433.246} C_VEL
LIN {X 0,Y 349.768,Z 567.262,A -85,B 0,C 180,E1 -22434.872,E2 -22434.872} C_VEL
LIN {X 0,Y 353.612,Z 554.829,A -85,B 0,C 180,E1 -22436.311,E2 -22436.311} C_VEL
LIN {X 0,Y 356.924,Z 542.525,A -85,B 0,C 180,E1 -22437.466,E2 -22437.466} C_VEL
LIN {X 0,Y 360.142,Z 528.986,A -85,B 0,C 180,E1 -22438.46,E2 -22438.46} C_VEL
LIN {X 0,Y 362.883,Z 515.212,A -85,B 0,C 180,E1 -22439.25,E2 -22439.25} C_VEL
LIN {X 0,Y 365.345,Z 499.781,A -85,B 0,C 180,E1 -22439.902,E2 -22439.902} C_VEL
LIN {X 0,Y 374.056,Z 418.682,A -85,B 0,C 180,E1 -22442.44,E2 -22442.44} C_VEL
LIN {X 0,Y 373.721,Z 399.897,A -85,B 0,C 180,E1 -22443.566,E2 -22443.566} C_VEL
LIN {X 0,Y 372.775,Z 384.023,A -85,B 0,C 180,E1 -22444.734,E2 -22444.734} C_VEL
LIN {X 0,Y 371.275,Z 378.531,A -85,B 0,C 180,E1 -22445.462,E2 -22445.462} C_VEL
LIN {X 0,Y 366.342,Z 370.61,A -85,B 0,C 180,E1 -22447.42,E2 -22447.42} C_VEL
LIN {X 0,Y 361.61,Z 363.874,A -85,B 0,C 180,E1 -22449.599,E2 -22449.599} C_VEL
LIN {X 0,Y 357.409,Z 358.336,A -85,B 0,C 180,E1 -22451.975,E2 -22451.975} C_VEL
LIN {X 0,Y 354.453,Z 354.82,A -85,B 0,C 180,E1 -22454.127,E2 -22454.127} C_VEL
LIN {X 0,Y 351.593,Z 351.391,A -85,B 0,C 180,E1 -22457.289,E2 -22457.289} C_VEL
LIN {X 0,Y 351.004,Z 350.38,A -85,B 0,C 180,E1 -22459.318,E2 -22459.318} C_VEL
LIN {X 0,Y 350.537,Z 350.434,A -85,B 0,C 180,E1 -22461.724,E2 -22461.724} C_VEL
LIN {X 0,Y 350.624,Z 351.219,A -85,B 0,C 180,E1 -22463.422,E2 -22463.422} C_VEL
LIN {X 0,Y 352.114,Z 353.728,A -85,B 0,C 180,E1 -22466.152,E2 -22466.152} C_VEL
LIN {X 0,Y 354.683,Z 357.42,A -85,B 0,C 180,E1 -22468.7,E2 -22468.7} C_VEL
LIN {X 0,Y 358.383,Z 363.143,A -85,B 0,C 180,E1 -22471.299,E2 -22471.299} C_VEL
LIN {X 0,Y 362.09,Z 369.347,A -85,B 0,C 180,E1 -22473.359,E2 -22473.359} C_VEL
LIN {X 0,Y 365.156,Z 374.708,A -85,B 0,C 180,E1 -22474.811,E2 -22474.811} C_VEL
LIN {X 0,Y 368.411,Z 380.92,A -85,B 0,C 180,E1 -22476.211,E2 -22476.211} C_VEL
LIN {X 0,Y 372.043,Z 388.629,A -85,B 0,C 180,E1 -22477.653,E2 -22477.653} C_VEL
LIN {X 0,Y 375.286,Z 396.783,A -85,B 0,C 180,E1 -22478.89,E2 -22478.89} C_VEL
LIN {X 0,Y 375.84,Z 403.734,A -85,B 0,C 180,E1 -22479.391,E2 -22479.391} C_VEL
LIN {X 0,Y 366.12,Z 491.66,A -85,B 0,C 180,E1 -22482.103,E2 -22482.103} C_VEL
LIN {X 0,Y 363.629,Z 507.656,A -85,B 0,C 180,E1 -22482.845,E2 -22482.845} C_VEL
LIN {X 0,Y 360.769,Z 522.538,A -85,B 0,C 180,E1 -22483.794,E2 -22483.794} C_VEL
LIN {X 0,Y 357.37,Z 536.605,A -85,B 0,C 180,E1 -22484.948,E2 -22484.948} C_VEL
LIN {X 0,Y 353.884,Z 549.294,A -85,B 0,C 180,E1 -22486.26,E2 -22486.26} C_VEL
LIN {X 0,Y 350.591,Z 559.829,A -85,B 0,C 180,E1 -22487.598,E2 -22487.598} C_VEL
LIN {X 0,Y 347.027,Z 570.39,A -85,B 0,C 180,E1 -22489.239,E2 -22489.239} C_VEL
LIN {X 0,Y 343.281,Z 580.478,A -85,B 0,C 180,E1 -22491.197,E2 -22491.197} C_VEL
LIN {X 0,Y 339.914,Z 588.761,A -85,B 0,C 180,E1 -22493.195,E2 -22493.195} C_VEL
LIN {X 0,Y 336.862,Z 595.492,A -85,B 0,C 180,E1 -22495.229,E2 -22495.229} C_VEL
LIN {X 0,Y 334.695,Z 600.11,A -85,B 0,C 180,E1 -22497.001,E2 -22497.001} C_VEL
LIN {X 0,Y 332.839,Z 603.827,A -85,B 0,C 180,E1 -22498.794,E2 -22498.794} C_VEL
LIN {X 0,Y 330.937,Z 607.42,A -85,B 0,C 180,E1 -22501.213,E2 -22501.213} C_VEL
LIN {X 0,Y 329.643,Z 609.575,A -85,B 0,C 180,E1 -22503.655,E2 -22503.655} C_VEL
LIN {X 0,Y 328.652,Z 610.354,A -85,B 0,C 180,E1 -22506.117,E2 -22506.117} C_VEL
LIN {X 0,Y 328.069,Z 609.721,A -85,B 0,C 180,E1 -22508.595,E2 -22508.595} C_VEL
LIN {X 0,Y 327.907,Z 608.042,A -85,B 0,C 180,E1 -22510.69,E2 -22510.69} C_VEL
LIN {X 0,Y 327.771,Z 605.029,A -85,B 0,C 180,E1 -22512.967,E2 -22512.967} C_VEL
LIN {X 0,Y 327.92,Z 601.516,A -85,B 0,C 180,E1 -22514.852,E2 -22514.852} C_VEL
LIN {X 0,Y 328.139,Z 596.987,A -85,B 0,C 180,E1 -22516.748,E2 -22516.748} C_VEL
LIN {X 0,Y 328.452,Z 590.212,A -85,B 0,C 180,E1 -22518.979,E2 -22518.979} C_VEL
LIN {X 0,Y 328.89,Z 582.687,A -85,B 0,C 180,E1 -22520.97,E2 -22520.97} C_VEL
LIN {X 0,Y 329.475,Z 574.156,A -85,B 0,C 180,E1 -22522.829,E2 -22522.829} C_VEL
LIN {X 0,Y 330.304,Z 563.316,A -85,B 0,C 180,E1 -22524.774,E2 -22524.774} C_VEL
LIN {X 0,Y 331.152,Z 552.447,A -85,B 0,C 180,E1 -22526.371,E2 -22526.371} C_VEL
LIN {X 0,Y 332.114,Z 540.578,A -85,B 0,C 180,E1 -22527.816,E2 -22527.816} C_VEL
LIN {X 0,Y 333.062,Z 527.693,A -85,B 0,C 180,E1 -22529.1,E2 -22529.1} C_VEL
LIN {X 0,Y 334.019,Z 513.652,A -85,B 0,C 180,E1 -22530.218,E2 -22530.218} C_VEL
LIN {X 0,Y 334.938,Z 498.866,A -85,B 0,C 180,E1 -22531.107,E2 -22531.107} C_VEL
LIN {X 0,Y 335.742,Z 483.577,A -85,B 0,C 180,E1 -22531.766,E2 -22531.766} C_VEL
LIN {X 0,Y 339.145,Z 384.478,A -85,B 0,C 180,E1 -22534.746,E2 -22534.746} C_VEL
LIN {X 0,Y 335.505,Z 351,A -85,B 0,C 180,E1 -22535.924,E2 -22535.924} C_VEL
LIN {X 0,Y 335.15,Z 345.723,A -85,B 0,C 180,E1 -22536.128,E2 -22536.128} C_VEL
LIN {X 0,Y 335.492,Z 339.438,A -85,B 0,C 180,E1 -22537.262,E2 -22537.262} C_VEL
LIN {X 0,Y 332.066,Z 322.257,A -85,B 0,C 180,E1 -22540.588,E2 -22540.588} C_VEL
LIN {X 0,Y 330.774,Z 315.841,A -85,B 0,C 180,E1 -22541.869,E2 -22541.869} C_VEL
LIN {X 0,Y 330.695,Z 315.845,A -85,B 0,C 180,E1 -22546.067,E2 -22546.067} C_VEL
LIN {X 0,Y 330.69,Z 315.848,A -85,B 0,C 180,E1 -22549.687,E2 -22549.687} C_VEL
LIN {X 0,Y 330.732,Z 315.846,A -85,B 0,C 180,E1 -22552.105,E2 -22552.105} C_VEL
LIN {X 0,Y 330.746,Z 315.834,A -85,B 0,C 180,E1 -22555.683,E2 -22555.683} C_VEL
LIN {X 0,Y 330.717,Z 315.845,A -85,B 0,C 180,E1 -22559.446,E2 -22559.446} C_VEL
LIN {X 0,Y 330.781,Z 315.835,A -85,B 0,C 180,E1 -22562.794,E2 -22562.794} C_VEL
LIN {X 0,Y 330.796,Z 315.839,A -85,B 0,C 180,E1 -22566.274,E2 -22566.274} C_VEL
LIN {X 0,Y 330.858,Z 315.828,A -85,B 0,C 180,E1 -22568.903,E2 -22568.903} C_VEL
LIN {X 0,Y 330.915,Z 315.818,A -85,B 0,C 180,E1 -22572.759,E2 -22572.759} C_VEL
LIN {X 0,Y 330.918,Z 315.823,A -85,B 0,C 180,E1 -22575.611,E2 -22575.611} C_VEL
LIN {X 0,Y 332.014,Z 318.842,A -85,B 0,C 180,E1 -22575.761,E2 -22575.761} C_VEL
LIN {X 0,Y 338.067,Z 333.46,A -85,B 0,C 180,E1 -22576.507,E2 -22576.507} C_VEL
LIN {X 0,Y 343.433,Z 349.487,A -85,B 0,C 180,E1 -22577.214,E2 -22577.214} C_VEL
LIN {X 0,Y 340.96,Z 449.44,A -85,B 0,C 180,E1 -22579.305,E2 -22579.305} C_VEL
LIN {X 0,Y 340.298,Z 463.736,A -85,B 0,C 180,E1 -22579.846,E2 -22579.846} C_VEL
LIN {X 0,Y 339.384,Z 478.045,A -85,B 0,C 180,E1 -22580.643,E2 -22580.643} C_VEL
LIN {X 0,Y 338.301,Z 489.921,A -85,B 0,C 180,E1 -22581.514,E2 -22581.514} C_VEL
LIN {X 0,Y 337.106,Z 501.091,A -85,B 0,C 180,E1 -22582.535,E2 -22582.535} C_VEL
LIN {X 0,Y 335.542,Z 512.852,A -85,B 0,C 180,E1 -22583.856,E2 -22583.856} C_VEL
LIN {X 0,Y 334.225,Z 524.499,A -85,B 0,C 180,E1 -22585.49,E2 -22585.49} C_VEL
LIN {X 0,Y 332.684,Z 534.976,A -85,B 0,C 180,E1 -22587.282,E2 -22587.282} C_VEL
LIN {X 0,Y 331.537,Z 543.602,A -85,B 0,C 180,E1 -22589.089,E2 -22589.089} C_VEL
LIN {X 0,Y 330.265,Z 551.917,A -85,B 0,C 180,E1 -22591.212,E2 -22591.212} C_VEL
LIN {X 0,Y 329.751,Z 558.379,A -85,B 0,C 180,E1 -22593.285,E2 -22593.285} C_VEL
LIN {X 0,Y 329.094,Z 563.858,A -85,B 0,C 180,E1 -22595.493,E2 -22595.493} C_VEL
LIN {X 0,Y 328.634,Z 567.405,A -85,B 0,C 180,E1 -22597.344,E2 -22597.344} C_VEL
LIN {X 0,Y 328.396,Z 570.874,A -85,B 0,C 180,E1 -22599.821,E2 -22599.821} C_VEL
LIN {X 0,Y 328.428,Z 572.177,A -85,B 0,C 180,E1 -22601.171,E2 -22601.171} C_VEL
LIN {X 0,Y 328.48,Z 573.482,A -85,B 0,C 180,E1 -22603.563,E2 -22603.563} C_VEL
LIN {X 0,Y 328.897,Z 573.506,A -85,B 0,C 180,E1 -22606.069,E2 -22606.069} C_VEL
LIN {X 0,Y 329.579,Z 572.159,A -85,B 0,C 180,E1 -22608.586,E2 -22608.586} C_VEL
LIN {X 0,Y 330.737,Z 569.394,A -85,B 0,C 180,E1 -22611.099,E2 -22611.099} C_VEL
LIN {X 0,Y 332.325,Z 565.118,A -85,B 0,C 180,E1 -22613.604,E2 -22613.604} C_VEL
LIN {X 0,Y 334.349,Z 559.193,A -85,B 0,C 180,E1 -22616.096,E2 -22616.096} C_VEL
LIN {X 0,Y 336.59,Z 552.43,A -85,B 0,C 180,E1 -22618.253,E2 -22618.253} C_VEL
LIN {X 0,Y 339.154,Z 543.903,A -85,B 0,C 180,E1 -22620.393,E2 -22620.393} C_VEL
LIN {X 0,Y 341.697,Z 534.933,A -85,B 0,C 180,E1 -22622.203,E2 -22622.203} C_VEL
LIN {X 0,Y 344.044,Z 525.977,A -85,B 0,C 180,E1 -22623.692,E2 -22623.692} C_VEL
LIN {X 0,Y 346.573,Z 515.209,A -85,B 0,C 180,E1 -22625.166,E2 -22625.166} C_VEL
LIN {X 0,Y 349.019,Z 503.307,A -85,B 0,C 180,E1 -22626.485,E2 -22626.485} C_VEL
LIN {X 0,Y 351.24,Z 490.276,A -85,B 0,C 180,E1 -22627.638,E2 -22627.638} C_VEL
LIN {X 0,Y 352.973,Z 476.484,A -85,B 0,C 180,E1 -22628.594,E2 -22628.594} C_VEL
LIN {X 0,Y 354.426,Z 462.398,A -85,B 0,C 180,E1 -22629.294,E2 -22629.294} C_VEL
LIN {X 0,Y 355.355,Z 448.05,A -85,B 0,C 180,E1 -22629.772,E2 -22629.772} C_VEL
LIN {X 0,Y 358.287,Z 367.902,A -85,B 0,C 180,E1 -22631.393,E2 -22631.393} C_VEL
LIN {X 0,Y 350.267,Z 350.664,A -85,B 0,C 180,E1 -22632.724,E2 -22632.724} C_VEL
LIN {X 0,Y 341.774,Z 334.737,A -85,B 0,C 180,E1 -22634.168,E2 -22634.168} C_VEL
LIN {X 0,Y 336.756,Z 326.325,A -85,B 0,C 180,E1 -22635.046,E2 -22635.046} C_VEL
LIN {X 0,Y 333.301,Z 320.649,A -85,B 0,C 180,E1 -22635.669,E2 -22635.669} C_VEL
LIN {X 0,Y 331.169,Z 317.635,A -85,B 0,C 180,E1 -22636.049,E2 -22636.049} C_VEL
LIN {X 0,Y 330.714,Z 315.839,A -85,B 0,C 180,E1 -22636.198,E2 -22636.198} C_VEL
LIN {X 0,Y 330.678,Z 315.849,A -85,B 0,C 180,E1 -22639.684,E2 -22639.684} C_VEL
LIN {X 0,Y 330.725,Z 315.843,A -85,B 0,C 180,E1 -22642.107,E2 -22642.107} C_VEL
LIN {X 0,Y 330.734,Z 315.82,A -85,B 0,C 180,E1 -22645.679,E2 -22645.679} C_VEL
LIN {X 0,Y 330.728,Z 315.836,A -85,B 0,C 180,E1 -22646.485,E2 -22646.485} C_VEL
LIN {X 0,Y 330.091,Z 315.934,A -85,B 0,C 180,E1 -22647.502,E2 -22647.502} C_VEL
LIN {X 0,Y 327.246,Z 316.295,A -85,B 0,C 180,E1 -22649.157,E2 -22649.157} C_VEL
LIN {X 0,Y 324.818,Z 316.588,A -85,B 0,C 180,E1 -22650.498,E2 -22650.498} C_VEL
LIN {X 0,Y 323.779,Z 316.708,A -85,B 0,C 180,E1 -22651.536,E2 -22651.536} C_VEL
LIN {X 0,Y 323.696,Z 316.713,A -85,B 0,C 180,E1 -22651.887,E2 -22651.887} C_VEL
LIN {X 0,Y 323.748,Z 316.707,A -85,B 0,C 180,E1 -22655.728,E2 -22655.728} C_VEL
LIN {X 0,Y 323.757,Z 316.709,A -85,B 0,C 180,E1 -22659.748,E2 -22659.748} C_VEL
LIN {X 0,Y 323.794,Z 316.703,A -85,B 0,C 180,E1 -22662.371,E2 -22662.371} C_VEL
LIN {X 0,Y 323.901,Z 316.681,A -85,B 0,C 180,E1 -22666.672,E2 -22666.672} C_VEL
LIN {X 0,Y 323.977,Z 316.669,A -85,B 0,C 180,E1 -22671.295,E2 -22671.295} C_VEL
LIN {X 0,Y 324.128,Z 316.668,A -85,B 0,C 180,E1 -22673.797,E2 -22673.797} C_VEL
LIN {X 0,Y 324.134,Z 316.654,A -85,B 0,C 180,E1 -22677.523,E2 -22677.523} C_VEL
LIN {X 0,Y 324.145,Z 316.646,A -85,B 0,C 180,E1 -22681.238,E2 -22681.238} C_VEL
LIN {X 0,Y 324.12,Z 316.668,A -85,B 0,C 180,E1 -22684.959,E2 -22684.959} C_VEL
LIN {X 0,Y 324.037,Z 316.657,A -85,B 0,C 180,E1 -22687.452,E2 -22687.452} C_VEL
LIN {X 0,Y 323.898,Z 316.684,A -85,B 0,C 180,E1 -22691.223,E2 -22691.223} C_VEL
LIN {X 0,Y 323.896,Z 316.683,A -85,B 0,C 180,E1 -22693.762,E2 -22693.762} C_VEL
LIN {X 0,Y 323.798,Z 316.688,A -85,B 0,C 180,E1 -22697.872,E2 -22697.872} C_VEL
LIN {X 0,Y 323.755,Z 316.7,A -85,B 0,C 180,E1 -22701.58,E2 -22701.58} C_VEL
LIN {X 0,Y 323.736,Z 316.717,A -85,B 0,C 180,E1 -22704.68,E2 -22704.68} C_VEL
LIN {X 0,Y 323.702,Z 316.722,A -85,B 0,C 180,E1 -22708.428,E2 -22708.428} C_VEL
LIN {X 0,Y 323.705,Z 316.722,A -85,B 0,C 180,E1 -22712.453,E2 -22712.453} C_VEL
LIN {X 0,Y 323.736,Z 316.674,A -85,B 0,C 180,E1 -22715.745,E2 -22715.745} C_VEL
LIN {X 0,Y 323.737,Z 316.718,A -85,B 0,C 180,E1 -22718.862,E2 -22718.862} C_VEL
LIN {X 0,Y 323.693,Z 316.717,A -85,B 0,C 180,E1 -22722.636,E2 -22722.636} C_VEL
LIN {X 0,Y 323.747,Z 316.832,A -85,B 0,C 180,E1 -22726.392,E2 -22726.392} C_VEL
LIN {X 0,Y 326.612,Z 326.721,A -85,B 0,C 180,E1 -22729.961,E2 -22729.961} C_VEL
LIN {X 0,Y 329.19,Z 336.061,A -85,B 0,C 180,E1 -22733.095,E2 -22733.095} C_VEL
LIN {X 0,Y 331.434,Z 345.637,A -85,B 0,C 180,E1 -22736.005,E2 -22736.005} C_VEL
LIN {X 0,Y 341.182,Z 366.046,A -85,B 0,C 180,E1 -22737.819,E2 -22737.819} C_VEL
LIN {X 0,Y 343.807,Z 372.11,A -85,B 0,C 180,E1 -22738.295,E2 -22738.295} C_VEL
LIN {X 0,Y 348.828,Z 402.201,A -85,B 0,C 180,E1 -22739.637,E2 -22739.637} C_VEL
LIN {X 0,Y 350.689,Z 417.733,A -85,B 0,C 180,E1 -22740.227,E2 -22740.227} C_VEL
LIN {X 0,Y 348.039,Z 485.049,A -85,B 0,C 180,E1 -22741.614,E2 -22741.614} C_VEL
LIN {X 0,Y 346.756,Z 499.449,A -85,B 0,C 180,E1 -22742.115,E2 -22742.115} C_VEL
LIN {X 0,Y 344.86,Z 513.319,A -85,B 0,C 180,E1 -22742.81,E2 -22742.81} C_VEL
LIN {X 0,Y 342.694,Z 525.389,A -85,B 0,C 180,E1 -22743.609,E2 -22743.609} C_VEL
LIN {X 0,Y 340.132,Z 538.111,A -85,B 0,C 180,E1 -22744.707,E2 -22744.707} C_VEL
LIN {X 0,Y 337.422,Z 549.81,A -85,B 0,C 180,E1 -22745.977,E2 -22745.977} C_VEL
LIN {X 0,Y 334.48,Z 561.328,A -85,B 0,C 180,E1 -22747.535,E2 -22747.535} C_VEL
LIN {X 0,Y 331.492,Z 571.761,A -85,B 0,C 180,E1 -22749.276,E2 -22749.276} C_VEL
LIN {X 0,Y 328.505,Z 581.708,A -85,B 0,C 180,E1 -22751.351,E2 -22751.351} C_VEL
LIN {X 0,Y 326.154,Z 589.769,A -85,B 0,C 180,E1 -22753.471,E2 -22753.471} C_VEL
LIN {X 0,Y 324.313,Z 596.308,A -85,B 0,C 180,E1 -22755.622,E2 -22755.622} C_VEL
LIN {X 0,Y 322.68,Z 602.158,A -85,B 0,C 180,E1 -22758.103,E2 -22758.103} C_VEL
LIN {X 0,Y 321.811,Z 605.563,A -85,B 0,C 180,E1 -22759.975,E2 -22759.975} C_VEL
LIN {X 0,Y 321.144,Z 608.804,A -85,B 0,C 180,E1 -22762.484,E2 -22762.484} C_VEL
LIN {X 0,Y 321.14,Z 610.711,A -85,B 0,C 180,E1 -22764.998,E2 -22764.998} C_VEL
LIN {X 0,Y 321.227,Z 611.29,A -85,B 0,C 180,E1 -22766.018,E2 -22766.018} C_VEL
LIN {X 0,Y 321.215,Z 615.768,A -85,B 0,C 180,E1 -22768.129,E2 -22768.129} C_VEL
LIN {X 0,Y 321.151,Z 618.724,A -85,B 0,C 180,E1 -22770.003,E2 -22770.003} C_VEL
LIN {X 0,Y 321.103,Z 620.212,A -85,B 0,C 180,E1 -22771.253,E2 -22771.253} C_VEL
LIN {X 0,Y 320.977,Z 622.055,A -85,B 0,C 180,E1 -22773.757,E2 -22773.757} C_VEL
LIN {X 0,Y 321.189,Z 622.478,A -85,B 0,C 180,E1 -22776.263,E2 -22776.263} C_VEL
LIN {X 0,Y 321.767,Z 621.522,A -85,B 0,C 180,E1 -22778.768,E2 -22778.768} C_VEL
LIN {X 0,Y 323.062,Z 619.196,A -85,B 0,C 180,E1 -22781.255,E2 -22781.255} C_VEL
LIN {X 0,Y 324.926,Z 615.456,A -85,B 0,C 180,E1 -22783.72,E2 -22783.72} C_VEL
LIN {X 0,Y 326.67,Z 611.691,A -85,B 0,C 180,E1 -22785.55,E2 -22785.55} C_VEL
LIN {X 0,Y 329.67,Z 605.206,A -85,B 0,C 180,E1 -22787.946,E2 -22787.946} C_VEL
LIN {X 0,Y 332.748,Z 598.066,A -85,B 0,C 180,E1 -22790.006,E2 -22790.006} C_VEL
LIN {X 0,Y 336.244,Z 589.374,A -85,B 0,C 180,E1 -22792.025,E2 -22792.025} C_VEL
LIN {X 0,Y 339.761,Z 580.347,A -85,B 0,C 180,E1 -22793.706,E2 -22793.706} C_VEL
LIN {X 0,Y 343.586,Z 569.65,A -85,B 0,C 180,E1 -22795.351,E2 -22795.351} C_VEL
LIN {X 0,Y 347.503,Z 557.726,A -85,B 0,C 180,E1 -22796.811,E2 -22796.811} C_VEL
LIN {X 0,Y 351.287,Z 544.682,A -85,B 0,C 180,E1 -22798.106,E2 -22798.106} C_VEL
LIN {X 0,Y 354.579,Z 531.845,A -85,B 0,C 180,E1 -22799.11,E2 -22799.11} C_VEL
LIN {X 0,Y 357.668,Z 517.853,A -85,B 0,C 180,E1 -22799.962,E2 -22799.962} C_VEL
LIN {X 0,Y 360.342,Z 502.641,A -85,B 0,C 180,E1 -22800.643,E2 -22800.643} C_VEL
LIN {X 0,Y 363.097,Z 478.957,A -85,B 0,C 180,E1 -22801.43,E2 -22801.43} C_VEL
LIN {X 0,Y 369.764,Z 419.897,A -85,B 0,C 180,E1 -22803.299,E2 -22803.299} C_VEL
LIN {X 0,Y 369.615,Z 401.912,A -85,B 0,C 180,E1 -22804.405,E2 -22804.405} C_VEL
LIN {X 0,Y 368.935,Z 387.652,A -85,B 0,C 180,E1 -22805.483,E2 -22805.483} C_VEL
LIN {X 0,Y 367.83,Z 383.626,A -85,B 0,C 180,E1 -22806.053,E2 -22806.053} C_VEL
LIN {X 0,Y 363.327,Z 376.243,A -85,B 0,C 180,E1 -22807.946,E2 -22807.946} C_VEL
LIN {X 0,Y 359.188,Z 370.129,A -85,B 0,C 180,E1 -22809.974,E2 -22809.974} C_VEL
LIN {X 0,Y 355.182,Z 364.675,A -85,B 0,C 180,E1 -22812.373,E2 -22812.373} C_VEL
LIN {X 0,Y 352.464,Z 361.379,A -85,B 0,C 180,E1 -22814.479,E2 -22814.479} C_VEL
LIN {X 0,Y 349.896,Z 358.173,A -85,B 0,C 180,E1 -22817.516,E2 -22817.516} C_VEL
LIN {X 0,Y 348.98,Z 357.15,A -85,B 0,C 180,E1 -22819.706,E2 -22819.706} C_VEL
LIN {X 0,Y 348.838,Z 357.592,A -85,B 0,C 180,E1 -22822.505,E2 -22822.505} C_VEL
LIN {X 0,Y 349.874,Z 359.651,A -85,B 0,C 180,E1 -22825.17,E2 -22825.17} C_VEL
LIN {X 0,Y 352.242,Z 363.195,A -85,B 0,C 180,E1 -22827.955,E2 -22827.955} C_VEL
LIN {X 0,Y 355.912,Z 369.053,A -85,B 0,C 180,E1 -22830.791,E2 -22830.791} C_VEL
LIN {X 0,Y 359.496,Z 375.363,A -85,B 0,C 180,E1 -22832.921,E2 -22832.921} C_VEL
LIN {X 0,Y 362.305,Z 380.491,A -85,B 0,C 180,E1 -22834.344,E2 -22834.344} C_VEL
LIN {X 0,Y 365.255,Z 386.388,A -85,B 0,C 180,E1 -22835.7,E2 -22835.7} C_VEL
LIN {X 0,Y 368.653,Z 393.863,A -85,B 0,C 180,E1 -22837.129,E2 -22837.129} C_VEL
LIN {X 0,Y 371.347,Z 401.039,A -85,B 0,C 180,E1 -22838.233,E2 -22838.233} C_VEL
LIN {X 0,Y 371.556,Z 405.65,A -85,B 0,C 180,E1 -22838.552,E2 -22838.552} C_VEL
LIN {X 0,Y 361.55,Z 491.824,A -85,B 0,C 180,E1 -22841.248,E2 -22841.248} C_VEL
LIN {X 0,Y 359.047,Z 507.182,A -85,B 0,C 180,E1 -22841.959,E2 -22841.959} C_VEL
LIN {X 0,Y 356.227,Z 521.25,A -85,B 0,C 180,E1 -22842.846,E2 -22842.846} C_VEL
LIN {X 0,Y 353.09,Z 534.179,A -85,B 0,C 180,E1 -22843.875,E2 -22843.875} C_VEL
LIN {X 0,Y 349.706,Z 546.053,A -85,B 0,C 180,E1 -22845.047,E2 -22845.047} C_VEL
LIN {X 0,Y 345.582,Z 558.908,A -85,B 0,C 180,E1 -22846.636,E2 -22846.636} C_VEL
LIN {X 0,Y 342.011,Z 569.009,A -85,B 0,C 180,E1 -22848.182,E2 -22848.182} C_VEL
LIN {X 0,Y 338.001,Z 579.399,A -85,B 0,C 180,E1 -22850.156,E2 -22850.156} C_VEL
LIN {X 0,Y 334.41,Z 587.858,A -85,B 0,C 180,E1 -22852.175,E2 -22852.175} C_VEL
LIN {X 0,Y 330.758,Z 595.503,A -85,B 0,C 180,E1 -22854.473,E2 -22854.473} C_VEL
LIN {X 0,Y 328.323,Z 600.281,A -85,B 0,C 180,E1 -22856.33,E2 -22856.33} C_VEL
LIN {X 0,Y 325.754,Z 605.041,A -85,B 0,C 180,E1 -22858.768,E2 -22858.768} C_VEL
LIN {X 0,Y 323.834,Z 608.284,A -85,B 0,C 180,E1 -22861.239,E2 -22861.239} C_VEL
LIN {X 0,Y 322.49,Z 610.1,A -85,B 0,C 180,E1 -22863.736,E2 -22863.736} C_VEL
LIN {X 0,Y 321.491,Z 610.517,A -85,B 0,C 180,E1 -22866.254,E2 -22866.254} C_VEL
LIN {X 0,Y 320.94,Z 609.519,A -85,B 0,C 180,E1 -22868.788,E2 -22868.788} C_VEL
LIN {X 0,Y 320.819,Z 607.825,A -85,B 0,C 180,E1 -22870.728,E2 -22870.728} C_VEL
LIN {X 0,Y 320.695,Z 604.225,A -85,B 0,C 180,E1 -22873.258,E2 -22873.258} C_VEL
LIN {X 0,Y 320.945,Z 599.23,A -85,B 0,C 180,E1 -22875.703,E2 -22875.703} C_VEL
LIN {X 0,Y 321.141,Z 593.674,A -85,B 0,C 180,E1 -22877.78,E2 -22877.78} C_VEL
LIN {X 0,Y 321.595,Z 585.981,A -85,B 0,C 180,E1 -22880.062,E2 -22880.062} C_VEL
LIN {X 0,Y 322.102,Z 577.778,A -85,B 0,C 180,E1 -22882.032,E2 -22882.032} C_VEL
LIN {X 0,Y 322.822,Z 567.775,A -85,B 0,C 180,E1 -22884.006,E2 -22884.006} C_VEL
LIN {X 0,Y 323.722,Z 556.591,A -85,B 0,C 180,E1 -22885.814,E2 -22885.814} C_VEL
LIN {X 0,Y 324.792,Z 543.672,A -85,B 0,C 180,E1 -22887.524,E2 -22887.524} C_VEL
LIN {X 0,Y 325.78,Z 530.484,A -85,B 0,C 180,E1 -22888.931,E2 -22888.931} C_VEL
LIN {X 0,Y 326.722,Z 517.059,A -85,B 0,C 180,E1 -22890.075,E2 -22890.075} C_VEL
LIN {X 0,Y 327.681,Z 502.705,A -85,B 0,C 180,E1 -22891.027,E2 -22891.027} C_VEL
LIN {X 0,Y 328.474,Z 488.557,A -85,B 0,C 180,E1 -22891.722,E2 -22891.722} C_VEL
LIN {X 0,Y 329.562,Z 455.985,A -85,B 0,C 180,E1 -22892.773,E2 -22892.773} C_VEL
LIN {X 0,Y 332.178,Z 385.161,A -85,B 0,C 180,E1 -22894.956,E2 -22894.956} C_VEL
LIN {X 0,Y 328.527,Z 351.045,A -85,B 0,C 180,E1 -22896.18,E2 -22896.18} C_VEL
LIN {X 0,Y 328.176,Z 345.935,A -85,B 0,C 180,E1 -22896.372,E2 -22896.372} C_VEL
LIN {X 0,Y 328.448,Z 340.158,A -85,B 0,C 180,E1 -22897.43,E2 -22897.43} C_VEL
LIN {X 0,Y 324.788,Z 322.07,A -85,B 0,C 180,E1 -22900.987,E2 -22900.987} C_VEL
LIN {X 0,Y 323.697,Z 316.724,A -85,B 0,C 180,E1 -22902.086,E2 -22902.086} C_VEL
LIN {X 0,Y 323.664,Z 316.722,A -85,B 0,C 180,E1 -22906.167,E2 -22906.167} C_VEL
LIN {X 0,Y 323.644,Z 316.725,A -85,B 0,C 180,E1 -22909.51,E2 -22909.51} C_VEL
LIN {X 0,Y 323.683,Z 316.72,A -85,B 0,C 180,E1 -22913.195,E2 -22913.195} C_VEL
LIN {X 0,Y 323.697,Z 316.711,A -85,B 0,C 180,E1 -22915.76,E2 -22915.76} C_VEL
LIN {X 0,Y 323.65,Z 316.727,A -85,B 0,C 180,E1 -22918.704,E2 -22918.704} C_VEL
LIN {X 0,Y 323.72,Z 316.712,A -85,B 0,C 180,E1 -22922.515,E2 -22922.515} C_VEL
LIN {X 0,Y 323.743,Z 316.716,A -85,B 0,C 180,E1 -22925.724,E2 -22925.724} C_VEL
LIN {X 0,Y 323.785,Z 316.711,A -85,B 0,C 180,E1 -22929.746,E2 -22929.746} C_VEL
LIN {X 0,Y 323.826,Z 316.704,A -85,B 0,C 180,E1 -22933.666,E2 -22933.666} C_VEL
LIN {X 0,Y 323.867,Z 316.7,A -85,B 0,C 180,E1 -22935.121,E2 -22935.121} C_VEL
LIN {X 0,Y 324.85,Z 319.522,A -85,B 0,C 180,E1 -22935.262,E2 -22935.262} C_VEL
LIN {X 0,Y 331.74,Z 335.77,A -85,B 0,C 180,E1 -22936.131,E2 -22936.131} C_VEL
LIN {X 0,Y 336.889,Z 351.658,A -85,B 0,C 180,E1 -22936.839,E2 -22936.839} C_VEL
LIN {X 0,Y 334.288,Z 449.008,A -85,B 0,C 180,E1 -22938.898,E2 -22938.898} C_VEL
LIN {X 0,Y 333.604,Z 462.87,A -85,B 0,C 180,E1 -22939.411,E2 -22939.411} C_VEL
LIN {X 0,Y 332.789,Z 476.373,A -85,B 0,C 180,E1 -22940.15,E2 -22940.15} C_VEL
LIN {X 0,Y 331.662,Z 488.704,A -85,B 0,C 180,E1 -22941.037,E2 -22941.037} C_VEL
LIN {X 0,Y 330.483,Z 500.169,A -85,B 0,C 180,E1 -22942.079,E2 -22942.079} C_VEL
LIN {X 0,Y 328.826,Z 512.173,A -85,B 0,C 180,E1 -22943.423,E2 -22943.423} C_VEL
LIN {X 0,Y 327.601,Z 522.087,A -85,B 0,C 180,E1 -22944.783,E2 -22944.783} C_VEL
LIN {X 0,Y 326.376,Z 531.349,A -85,B 0,C 180,E1 -22946.306,E2 -22946.306} C_VEL
LIN {X 0,Y 324.923,Z 540.694,A -85,B 0,C 180,E1 -22948.144,E2 -22948.144} C_VEL
LIN {X 0,Y 323.834,Z 548.438,A -85,B 0,C 180,E1 -22949.997,E2 -22949.997} C_VEL
LIN {X 0,Y 323.029,Z 554.869,A -85,B 0,C 180,E1 -22951.861,E2 -22951.861} C_VEL
LIN {X 0,Y 322.515,Z 560.202,A -85,B 0,C 180,E1 -22953.733,E2 -22953.733} C_VEL
LIN {X 0,Y 321.795,Z 565.863,A -85,B 0,C 180,E1 -22956.245,E2 -22956.245} C_VEL
LIN {X 0,Y 321.362,Z 569.977,A -85,B 0,C 180,E1 -22958.773,E2 -22958.773} C_VEL
LIN {X 0,Y 321.352,Z 572.638,A -85,B 0,C 180,E1 -22961.31,E2 -22961.31} C_VEL
LIN {X 0,Y 321.426,Z 573.93,A -85,B 0,C 180,E1 -22963.866,E2 -22963.866} C_VEL
LIN {X 0,Y 321.914,Z 573.862,A -85,B 0,C 180,E1 -22966.428,E2 -22966.428} C_VEL
LIN {X 0,Y 322.658,Z 572.428,A -85,B 0,C 180,E1 -22969,E2 -22969} C_VEL
LIN {X 0,Y 323.927,Z 569.532,A -85,B 0,C 180,E1 -22971.594,E2 -22971.594} C_VEL
LIN {X 0,Y 325.591,Z 565.201,A -85,B 0,C 180,E1 -22974.122,E2 -22974.122} C_VEL
LIN {X 0,Y 327.049,Z 561.126,A -85,B 0,C 180,E1 -22975.905,E2 -22975.905} C_VEL
LIN {X 0,Y 329.418,Z 554.361,A -85,B 0,C 180,E1 -22978.232,E2 -22978.232} C_VEL
LIN {X 0,Y 331.499,Z 548.065,A -85,B 0,C 180,E1 -22979.967,E2 -22979.967} C_VEL
LIN {X 0,Y 334.123,Z 539.246,A -85,B 0,C 180,E1 -22981.956,E2 -22981.956} C_VEL
LIN {X 0,Y 336.827,Z 529.598,A -85,B 0,C 180,E1 -22983.714,E2 -22983.714} C_VEL
LIN {X 0,Y 339.532,Z 519.025,A -85,B 0,C 180,E1 -22985.28,E2 -22985.28} C_VEL
LIN {X 0,Y 342.075,Z 507.622,A -85,B 0,C 180,E1 -22986.655,E2 -22986.655} C_VEL
LIN {X 0,Y 344.281,Z 495.933,A -85,B 0,C 180,E1 -22987.795,E2 -22987.795} C_VEL
LIN {X 0,Y 346.265,Z 482.616,A -85,B 0,C 180,E1 -22988.831,E2 -22988.831} C_VEL
LIN {X 0,Y 347.711,Z 470.169,A -85,B 0,C 180,E1 -22989.569,E2 -22989.569} C_VEL
LIN {X 0,Y 348.98,Z 455.618,A -85,B 0,C 180,E1 -22990.18,E2 -22990.18} C_VEL
LIN {X 0,Y 349.696,Z 440.87,A -85,B 0,C 180,E1 -22990.567,E2 -22990.567} C_VEL
LIN {X 0,Y 352.376,Z 370.05,A -85,B 0,C 180,E1 -22992,E2 -22992} C_VEL
LIN {X 0,Y 344.735,Z 353.677,A -85,B 0,C 180,E1 -22993.31,E2 -22993.31} C_VEL
LIN {X 0,Y 336.874,Z 338.821,A -85,B 0,C 180,E1 -22994.697,E2 -22994.697} C_VEL
LIN {X 0,Y 332.203,Z 330.933,A -85,B 0,C 180,E1 -22995.54,E2 -22995.54} C_VEL
LIN {X 0,Y 327.92,Z 324.351,A -85,B 0,C 180,E1 -22996.325,E2 -22996.325} C_VEL
LIN {X 0,Y 325.86,Z 320.991,A -85,B 0,C 180,E1 -22996.719,E2 -22996.719} C_VEL
LIN {X 0,Y 324.137,Z 318.553,A -85,B 0,C 180,E1 -22997.045,E2 -22997.045} C_VEL
LIN {X 0,Y 323.671,Z 316.725,A -85,B 0,C 180,E1 -22997.188,E2 -22997.188} C_VEL
LIN {X 0,Y 323.684,Z 316.723,A -85,B 0,C 180,E1 -23001.166,E2 -23001.166} C_VEL
LIN {X 0,Y 323.708,Z 316.689,A -85,B 0,C 180,E1 -23005.304,E2 -23005.304} C_VEL
LIN {X 0,Y 323.669,Z 316.716,A -85,B 0,C 180,E1 -23008.709,E2 -23008.709} C_VEL
LIN {X 0,Y 323.696,Z 316.713,A -85,B 0,C 180,E1 -23011.887,E2 -23011.887} C_VEL
LIN {X 0,Y 323.032,Z 316.795,A -85,B 0,C 180,E1 -23012.926,E2 -23012.926} C_VEL
LIN {X 0,Y 320.174,Z 317.161,A -85,B 0,C 180,E1 -23014.616,E2 -23014.616} C_VEL
LIN {X 0,Y 317.759,Z 317.452,A -85,B 0,C 180,E1 -23015.986,E2 -23015.986} C_VEL
LIN {X 0,Y 316.738,Z 317.574,A -85,B 0,C 180,E1 -23017.047,E2 -23017.047} C_VEL
LIN {X 0,Y 316.664,Z 317.585,A -85,B 0,C 180,E1 -23017.406,E2 -23017.406} C_VEL
LIN {X 0,Y 316.689,Z 317.581,A -85,B 0,C 180,E1 -23020.624,E2 -23020.624} C_VEL
LIN {X 0,Y 316.733,Z 317.582,A -85,B 0,C 180,E1 -23024.611,E2 -23024.611} C_VEL
LIN {X 0,Y 316.87,Z 317.562,A -85,B 0,C 180,E1 -23027.229,E2 -23027.229} C_VEL
LIN {X 0,Y 316.92,Z 317.547,A -85,B 0,C 180,E1 -23031.1,E2 -23031.1} C_VEL
LIN {X 0,Y 317.1,Z 317.544,A -85,B 0,C 180,E1 -23033.688,E2 -23033.688} C_VEL
LIN {X 0,Y 317.089,Z 317.53,A -85,B 0,C 180,E1 -23037.468,E2 -23037.468} C_VEL
LIN {X 0,Y 317.123,Z 317.52,A -85,B 0,C 180,E1 -23041.266,E2 -23041.266} C_VEL
LIN {X 0,Y 317.07,Z 317.545,A -85,B 0,C 180,E1 -23045.07,E2 -23045.07} C_VEL
LIN {X 0,Y 316.976,Z 317.537,A -85,B 0,C 180,E1 -23047.619,E2 -23047.619} C_VEL
LIN {X 0,Y 316.848,Z 317.56,A -85,B 0,C 180,E1 -23051.476,E2 -23051.476} C_VEL
LIN {X 0,Y 316.83,Z 317.568,A -85,B 0,C 180,E1 -23054.075,E2 -23054.075} C_VEL
LIN {X 0,Y 316.756,Z 317.566,A -85,B 0,C 180,E1 -23058.049,E2 -23058.049} C_VEL
LIN {X 0,Y 316.688,Z 317.578,A -85,B 0,C 180,E1 -23062.086,E2 -23062.086} C_VEL
LIN {X 0,Y 316.679,Z 317.583,A -85,B 0,C 180,E1 -23066.255,E2 -23066.255} C_VEL
LIN {X 0,Y 316.633,Z 317.59,A -85,B 0,C 180,E1 -23070.382,E2 -23070.382} C_VEL
LIN {X 0,Y 316.666,Z 317.581,A -85,B 0,C 180,E1 -23073.572,E2 -23073.572} C_VEL
LIN {X 0,Y 316.705,Z 317.562,A -85,B 0,C 180,E1 -23077.238,E2 -23077.238} C_VEL
LIN {X 0,Y 316.669,Z 317.596,A -85,B 0,C 180,E1 -23081.237,E2 -23081.237} C_VEL
LIN {X 0,Y 316.668,Z 317.66,A -85,B 0,C 180,E1 -23085.395,E2 -23085.395} C_VEL
LIN {X 0,Y 319.661,Z 327.744,A -85,B 0,C 180,E1 -23089.211,E2 -23089.211} C_VEL
LIN {X 0,Y 322.288,Z 337.361,A -85,B 0,C 180,E1 -23092.521,E2 -23092.521} C_VEL
LIN {X 0,Y 324.156,Z 345.027,A -85,B 0,C 180,E1 -23094.962,E2 -23094.962} C_VEL
LIN {X 0,Y 326.385,Z 349.44,A -85,B 0,C 180,E1 -23095.406,E2 -23095.406} C_VEL
LIN {X 0,Y 335.382,Z 368.253,A -85,B 0,C 180,E1 -23097.14,E2 -23097.14} C_VEL
LIN {X 0,Y 338.397,Z 375.29,A -85,B 0,C 180,E1 -23097.711,E2 -23097.711} C_VEL
LIN {X 0,Y 343.111,Z 404.208,A -85,B 0,C 180,E1 -23099.027,E2 -23099.027} C_VEL
LIN {X 0,Y 344.769,Z 417.472,A -85,B 0,C 180,E1 -23099.554,E2 -23099.554} C_VEL
LIN {X 0,Y 342.133,Z 484.194,A -85,B 0,C 180,E1 -23100.953,E2 -23100.953} C_VEL
LIN {X 0,Y 340.826,Z 498.746,A -85,B 0,C 180,E1 -23101.461,E2 -23101.461} C_VEL
LIN {X 0,Y 338.761,Z 513.253,A -85,B 0,C 180,E1 -23102.195,E2 -23102.195} C_VEL
LIN {X 0,Y 336.378,Z 526.122,A -85,B 0,C 180,E1 -23103.074,E2 -23103.074} C_VEL
LIN {X 0,Y 333.763,Z 538.621,A -85,B 0,C 180,E1 -23104.189,E2 -23104.189} C_VEL
LIN {X 0,Y 331.022,Z 549.931,A -85,B 0,C 180,E1 -23105.45,E2 -23105.45} C_VEL
LIN {X 0,Y 327.943,Z 561.547,A -85,B 0,C 180,E1 -23107.062,E2 -23107.062} C_VEL
LIN {X 0,Y 324.868,Z 571.87,A -85,B 0,C 180,E1 -23108.833,E2 -23108.833} C_VEL
LIN {X 0,Y 322.221,Z 580.422,A -85,B 0,C 180,E1 -23110.643,E2 -23110.643} C_VEL
LIN {X 0,Y 319.637,Z 588.659,A -85,B 0,C 180,E1 -23112.796,E2 -23112.796} C_VEL
LIN {X 0,Y 317.407,Z 596.144,A -85,B 0,C 180,E1 -23115.302,E2 -23115.302} C_VEL
LIN {X 0,Y 315.827,Z 601.409,A -85,B 0,C 180,E1 -23117.57,E2 -23117.57} C_VEL
LIN {X 0,Y 314.786,Z 605.285,A -85,B 0,C 180,E1 -23119.749,E2 -23119.749} C_VEL
LIN {X 0,Y 314.077,Z 608.475,A -85,B 0,C 180,E1 -23122.313,E2 -23122.313} C_VEL
LIN {X 0,Y 314.06,Z 610.333,A -85,B 0,C 180,E1 -23124.885,E2 -23124.885} C_VEL
LIN {X 0,Y 314.188,Z 610.929,A -85,B 0,C 180,E1 -23126.168,E2 -23126.168} C_VEL
LIN {X 0,Y 314.168,Z 615.01,A -85,B 0,C 180,E1 -23128.087,E2 -23128.087} C_VEL
LIN {X 0,Y 314.078,Z 618.09,A -85,B 0,C 180,E1 -23130.003,E2 -23130.003} C_VEL
LIN {X 0,Y 314.045,Z 619.662,A -85,B 0,C 180,E1 -23131.281,E2 -23131.281} C_VEL
LIN {X 0,Y 313.899,Z 621.695,A -85,B 0,C 180,E1 -23133.841,E2 -23133.841} C_VEL
LIN {X 0,Y 314.12,Z 622.325,A -85,B 0,C 180,E1 -23136.404,E2 -23136.404} C_VEL
LIN {X 0,Y 314.757,Z 621.578,A -85,B 0,C 180,E1 -23138.965,E2 -23138.965} C_VEL
LIN {X 0,Y 316.09,Z 619.461,A -85,B 0,C 180,E1 -23141.507,E2 -23141.507} C_VEL
LIN {X 0,Y 318.053,Z 615.926,A -85,B 0,C 180,E1 -23144.022,E2 -23144.022} C_VEL
LIN {X 0,Y 320.564,Z 610.928,A -85,B 0,C 180,E1 -23146.505,E2 -23146.505} C_VEL
LIN {X 0,Y 323.886,Z 604.303,A -85,B 0,C 180,E1 -23148.932,E2 -23148.932} C_VEL
LIN {X 0,Y 327.198,Z 597.046,A -85,B 0,C 180,E1 -23151.015,E2 -23151.015} C_VEL
LIN {X 0,Y 330.977,Z 588.205,A -85,B 0,C 180,E1 -23153.052,E2 -23153.052} C_VEL
LIN {X 0,Y 334.764,Z 579.016,A -85,B 0,C 180,E1 -23154.741,E2 -23154.741} C_VEL
LIN {X 0,Y 338.798,Z 568.083,A -85,B 0,C 180,E1 -23156.394,E2 -23156.394} C_VEL
LIN {X 0,Y 342.931,Z 555.96,A -85,B 0,C 180,E1 -23157.857,E2 -23157.857} C_VEL
LIN {X 0,Y 346.936,Z 542.679,A -85,B 0,C 180,E1 -23159.151,E2 -23159.151} C_VEL
LIN {X 0,Y 350.436,Z 529.439,A -85,B 0,C 180,E1 -23160.148,E2 -23160.148} C_VEL
LIN {X 0,Y 353.663,Z 514.833,A -85,B 0,C 180,E1 -23160.996,E2 -23160.996} C_VEL
LIN {X 0,Y 356.437,Z 498.952,A -85,B 0,C 180,E1 -23161.675,E2 -23161.675} C_VEL
LIN {X 0,Y 365.626,Z 421.358,A -85,B 0,C 180,E1 -23164.175,E2 -23164.175} C_VEL
LIN {X 0,Y 365.684,Z 404.025,A -85,B 0,C 180,E1 -23165.266,E2 -23165.266} C_VEL
LIN {X 0,Y 365.229,Z 391.299,A -85,B 0,C 180,E1 -23166.256,E2 -23166.256} C_VEL
LIN {X 0,Y 364.531,Z 388.811,A -85,B 0,C 180,E1 -23166.629,E2 -23166.629} C_VEL
LIN {X 0,Y 360.471,Z 381.984,A -85,B 0,C 180,E1 -23168.451,E2 -23168.451} C_VEL
LIN {X 0,Y 356.816,Z 376.424,A -85,B 0,C 180,E1 -23170.338,E2 -23170.338} C_VEL
LIN {X 0,Y 353.146,Z 371.29,A -85,B 0,C 180,E1 -23172.656,E2 -23172.656} C_VEL
LIN {X 0,Y 350.838,Z 368.316,A -85,B 0,C 180,E1 -23174.523,E2 -23174.523} C_VEL
LIN {X 0,Y 348.26,Z 364.999,A -85,B 0,C 180,E1 -23177.679,E2 -23177.679} C_VEL
LIN {X 0,Y 347.364,Z 364.011,A -85,B 0,C 180,E1 -23180.022,E2 -23180.022} C_VEL
LIN {X 0,Y 347.356,Z 364.706,A -85,B 0,C 180,E1 -23182.775,E2 -23182.775} C_VEL
LIN {X 0,Y 348.528,Z 366.947,A -85,B 0,C 180,E1 -23185.489,E2 -23185.489} C_VEL
LIN {X 0,Y 350.958,Z 370.86,A -85,B 0,C 180,E1 -23188.264,E2 -23188.264} C_VEL
LIN {X 0,Y 354.024,Z 376.072,A -85,B 0,C 180,E1 -23190.662,E2 -23190.662} C_VEL
LIN {X 0,Y 357.018,Z 381.525,A -85,B 0,C 180,E1 -23192.526,E2 -23192.526} C_VEL
LIN {X 0,Y 359.615,Z 386.489,A -85,B 0,C 180,E1 -23193.917,E2 -23193.917} C_VEL
LIN {X 0,Y 362.942,Z 393.452,A -85,B 0,C 180,E1 -23195.522,E2 -23195.522} C_VEL
LIN {X 0,Y 365.937,Z 400.902,A -85,B 0,C 180,E1 -23196.882,E2 -23196.882} C_VEL
LIN {X 0,Y 367.422,Z 404.969,A -85,B 0,C 180,E1 -23197.52,E2 -23197.52} C_VEL
LIN {X 0,Y 367.453,Z 407.556,A -85,B 0,C 180,E1 -23197.69,E2 -23197.69} C_VEL
LIN {X 0,Y 357.146,Z 492,A -85,B 0,C 180,E1 -23200.359,E2 -23200.359} C_VEL
LIN {X 0,Y 354.608,Z 506.92,A -85,B 0,C 180,E1 -23201.054,E2 -23201.054} C_VEL
LIN {X 0,Y 351.433,Z 521.93,A -85,B 0,C 180,E1 -23202.005,E2 -23202.005} C_VEL
LIN {X 0,Y 348.147,Z 534.744,A -85,B 0,C 180,E1 -23203.038,E2 -23203.038} C_VEL
LIN {X 0,Y 344.61,Z 546.557,A -85,B 0,C 180,E1 -23204.225,E2 -23204.225} C_VEL
LIN {X 0,Y 340.565,Z 558.537,A -85,B 0,C 180,E1 -23205.711,E2 -23205.711} C_VEL
LIN {X 0,Y 336.528,Z 569.342,A -85,B 0,C 180,E1 -23207.376,E2 -23207.376} C_VEL
LIN {X 0,Y 332.312,Z 579.683,A -85,B 0,C 180,E1 -23209.372,E2 -23209.372} C_VEL
LIN {X 0,Y 328.479,Z 588.114,A -85,B 0,C 180,E1 -23211.415,E2 -23211.415} C_VEL
LIN {X 0,Y 325.499,Z 594.118,A -85,B 0,C 180,E1 -23213.203,E2 -23213.203} C_VEL
LIN {X 0,Y 321.998,Z 600.498,A -85,B 0,C 180,E1 -23215.633,E2 -23215.633} C_VEL
LIN {X 0,Y 319.896,Z 604.195,A -85,B 0,C 180,E1 -23217.49,E2 -23217.49} C_VEL
LIN {X 0,Y 317.549,Z 607.781,A -85,B 0,C 180,E1 -23220,E2 -23220} C_VEL
LIN {X 0,Y 315.975,Z 609.927,A -85,B 0,C 180,E1 -23222.541,E2 -23222.541} C_VEL
LIN {X 0,Y 314.775,Z 610.71,A -85,B 0,C 180,E1 -23225.107,E2 -23225.107} C_VEL
LIN {X 0,Y 313.999,Z 610.099,A -85,B 0,C 180,E1 -23227.692,E2 -23227.692} C_VEL
LIN {X 0,Y 313.737,Z 608.065,A -85,B 0,C 180,E1 -23230.289,E2 -23230.289} C_VEL
LIN {X 0,Y 313.6,Z 604.467,A -85,B 0,C 180,E1 -23232.906,E2 -23232.906} C_VEL
LIN {X 0,Y 313.757,Z 600.723,A -85,B 0,C 180,E1 -23234.876,E2 -23234.876} C_VEL
LIN {X 0,Y 313.987,Z 595.877,A -85,B 0,C 180,E1 -23236.858,E2 -23236.858} C_VEL
LIN {X 0,Y 314.316,Z 588.75,A -85,B 0,C 180,E1 -23239.19,E2 -23239.19} C_VEL
LIN {X 0,Y 314.802,Z 581.139,A -85,B 0,C 180,E1 -23241.196,E2 -23241.196} C_VEL
LIN {X 0,Y 315.406,Z 571.814,A -85,B 0,C 180,E1 -23243.215,E2 -23243.215} C_VEL
LIN {X 0,Y 316.35,Z 560.466,A -85,B 0,C 180,E1 -23245.228,E2 -23245.228} C_VEL
LIN {X 0,Y 317.275,Z 548.918,A -85,B 0,C 180,E1 -23246.909,E2 -23246.909} C_VEL
LIN {X 0,Y 318.353,Z 535.456,A -85,B 0,C 180,E1 -23248.497,E2 -23248.497} C_VEL
LIN {X 0,Y 319.36,Z 522.255,A -85,B 0,C 180,E1 -23249.751,E2 -23249.751} C_VEL
LIN {X 0,Y 320.319,Z 507.86,A -85,B 0,C 180,E1 -23250.831,E2 -23250.831} C_VEL
LIN {X 0,Y 321.161,Z 492.75,A -85,B 0,C 180,E1 -23251.669,E2 -23251.669} C_VEL
LIN {X 0,Y 321.847,Z 477.467,A -85,B 0,C 180,E1 -23252.26,E2 -23252.26} C_VEL
LIN {X 0,Y 325.131,Z 385.512,A -85,B 0,C 180,E1 -23255.176,E2 -23255.176} C_VEL
LIN {X 0,Y 321.645,Z 352.203,A -85,B 0,C 180,E1 -23256.403,E2 -23256.403} C_VEL
LIN {X 0,Y 321.238,Z 345.959,A -85,B 0,C 180,E1 -23256.652,E2 -23256.652} C_VEL
LIN {X 0,Y 321.514,Z 341.921,A -85,B 0,C 180,E1 -23257.399,E2 -23257.399} C_VEL
LIN {X 0,Y 318.322,Z 325.761,A -85,B 0,C 180,E1 -23260.607,E2 -23260.607} C_VEL
LIN {X 0,Y 316.678,Z 317.599,A -85,B 0,C 180,E1 -23262.275,E2 -23262.275} C_VEL
LIN {X 0,Y 316.621,Z 317.603,A -85,B 0,C 180,E1 -23266.698,E2 -23266.698} C_VEL
LIN {X 0,Y 316.602,Z 317.604,A -85,B 0,C 180,E1 -23270.745,E2 -23270.745} C_VEL
LIN {X 0,Y 316.633,Z 317.599,A -85,B 0,C 180,E1 -23273.321,E2 -23273.321} C_VEL
LIN {X 0,Y 316.624,Z 317.592,A -85,B 0,C 180,E1 -23276.42,E2 -23276.42} C_VEL
LIN {X 0,Y 316.629,Z 317.601,A -85,B 0,C 180,E1 -23279.627,E2 -23279.627} C_VEL
LIN {X 0,Y 316.689,Z 317.592,A -85,B 0,C 180,E1 -23283.743,E2 -23283.743} C_VEL
LIN {X 0,Y 316.713,Z 317.592,A -85,B 0,C 180,E1 -23287.913,E2 -23287.913} C_VEL
LIN {X 0,Y 316.776,Z 317.583,A -85,B 0,C 180,E1 -23291.964,E2 -23291.964} C_VEL
LIN {X 0,Y 316.819,Z 317.748,A -85,B 0,C 180,E1 -23294.612,E2 -23294.612} C_VEL
LIN {X 0,Y 318.336,Z 321.677,A -85,B 0,C 180,E1 -23294.825,E2 -23294.825} C_VEL
LIN {X 0,Y 325.44,Z 338.181,A -85,B 0,C 180,E1 -23295.745,E2 -23295.745} C_VEL
LIN {X 0,Y 330.09,Z 352.193,A -85,B 0,C 180,E1 -23296.397,E2 -23296.397} C_VEL
LIN {X 0,Y 327.589,Z 449.747,A -85,B 0,C 180,E1 -23298.512,E2 -23298.512} C_VEL
LIN {X 0,Y 326.883,Z 463.484,A -85,B 0,C 180,E1 -23299.034,E2 -23299.034} C_VEL
LIN {X 0,Y 326.042,Z 476.933,A -85,B 0,C 180,E1 -23299.788,E2 -23299.788} C_VEL
LIN {X 0,Y 324.879,Z 489.232,A -85,B 0,C 180,E1 -23300.691,E2 -23300.691} C_VEL
LIN {X 0,Y 323.641,Z 500.681,A -85,B 0,C 180,E1 -23301.753,E2 -23301.753} C_VEL
LIN {X 0,Y 321.953,Z 512.664,A -85,B 0,C 180,E1 -23303.125,E2 -23303.125} C_VEL
LIN {X 0,Y 320.6,Z 523.526,A -85,B 0,C 180,E1 -23304.669,E2 -23304.669} C_VEL
LIN {X 0,Y 319.273,Z 532.662,A -85,B 0,C 180,E1 -23306.223,E2 -23306.223} C_VEL
LIN {X 0,Y 317.848,Z 541.832,A -85,B 0,C 180,E1 -23308.103,E2 -23308.103} C_VEL
LIN {X 0,Y 316.683,Z 549.478,A -85,B 0,C 180,E1 -23309.997,E2 -23309.997} C_VEL
LIN {X 0,Y 315.956,Z 555.815,A -85,B 0,C 180,E1 -23311.903,E2 -23311.903} C_VEL
LIN {X 0,Y 315.41,Z 561.045,A -85,B 0,C 180,E1 -23313.817,E2 -23313.817} C_VEL
LIN {X 0,Y 314.682,Z 566.611,A -85,B 0,C 180,E1 -23316.387,E2 -23316.387} C_VEL
LIN {X 0,Y 314.264,Z 570.618,A -85,B 0,C 180,E1 -23318.973,E2 -23318.973} C_VEL
LIN {X 0,Y 314.251,Z 573.169,A -85,B 0,C 180,E1 -23321.569,E2 -23321.569} C_VEL
LIN {X 0,Y 314.367,Z 574.374,A -85,B 0,C 180,E1 -23324.184,E2 -23324.184} C_VEL
LIN {X 0,Y 314.914,Z 574.219,A -85,B 0,C 180,E1 -23326.804,E2 -23326.804} C_VEL
LIN {X 0,Y 315.749,Z 572.698,A -85,B 0,C 180,E1 -23329.432,E2 -23329.432} C_VEL
LIN {X 0,Y 317.099,Z 569.752,A -85,B 0,C 180,E1 -23332.052,E2 -23332.052} C_VEL
LIN {X 0,Y 318.887,Z 565.288,A -85,B 0,C 180,E1 -23334.663,E2 -23334.663} C_VEL
LIN {X 0,Y 320.625,Z 560.637,A -85,B 0,C 180,E1 -23336.668,E2 -23336.668} C_VEL
LIN {X 0,Y 322.961,Z 554.241,A -85,B 0,C 180,E1 -23338.849,E2 -23338.849} C_VEL
LIN {X 0,Y 325.692,Z 546.026,A -85,B 0,C 180,E1 -23341.07,E2 -23341.07} C_VEL
LIN {X 0,Y 328.385,Z 537.336,A -85,B 0,C 180,E1 -23342.946,E2 -23342.946} C_VEL
LIN {X 0,Y 331.067,Z 527.928,A -85,B 0,C 180,E1 -23344.607,E2 -23344.607} C_VEL
LIN {X 0,Y 333.816,Z 517.127,A -85,B 0,C 180,E1 -23346.163,E2 -23346.163} C_VEL
LIN {X 0,Y 336.418,Z 505.634,A -85,B 0,C 180,E1 -23347.502,E2 -23347.502} C_VEL
LIN {X 0,Y 338.495,Z 494.577,A -85,B 0,C 180,E1 -23348.558,E2 -23348.558} C_VEL
LIN {X 0,Y 340.394,Z 481.776,A -85,B 0,C 180,E1 -23349.535,E2 -23349.535} C_VEL
LIN {X 0,Y 341.995,Z 468.147,A -85,B 0,C 180,E1 -23350.317,E2 -23350.317} C_VEL
LIN {X 0,Y 343.128,Z 454.614,A -85,B 0,C 180,E1 -23350.865,E2 -23350.865} C_VEL
LIN {X 0,Y 343.957,Z 435.625,A -85,B 0,C 180,E1 -23351.334,E2 -23351.334} C_VEL
LIN {X 0,Y 346.434,Z 372.014,A -85,B 0,C 180,E1 -23352.641,E2 -23352.641} C_VEL
LIN {X 0,Y 338.783,Z 355.675,A -85,B 0,C 180,E1 -23354.003,E2 -23354.003} C_VEL
LIN {X 0,Y 329.718,Z 338.803,A -85,B 0,C 180,E1 -23355.669,E2 -23355.669} C_VEL
LIN {X 0,Y 321.3,Z 325.688,A -85,B 0,C 180,E1 -23357.267,E2 -23357.267} C_VEL
LIN {X 0,Y 318.793,Z 321.908,A -85,B 0,C 180,E1 -23357.765,E2 -23357.765} C_VEL
LIN {X 0,Y 317.02,Z 319.292,A -85,B 0,C 180,E1 -23358.122,E2 -23358.122} C_VEL
LIN {X 0,Y 316.604,Z 317.602,A -85,B 0,C 180,E1 -23358.257,E2 -23358.257} C_VEL
LIN {X 0,Y 316.626,Z 317.604,A -85,B 0,C 180,E1 -23361.726,E2 -23361.726} C_VEL
LIN {X 0,Y 316.643,Z 317.565,A -85,B 0,C 180,E1 -23364.926,E2 -23364.926} C_VEL
LIN {X 0,Y 316.628,Z 317.6,A -85,B 0,C 180,E1 -23367.932,E2 -23367.932} C_VEL
LIN {X 0,Y 316.662,Z 317.587,A -85,B 0,C 180,E1 -23372.217,E2 -23372.217} C_VEL
LIN {X 0,Y 316.68,Z 317.595,A -85,B 0,C 180,E1 -23375.15,E2 -23375.15} C_VEL
LIN {X 0,Y 316.664,Z 317.585,A -85,B 0,C 180,E1 -23377.406,E2 -23377.406} C_VEL
LIN {X 0,Y 316.029,Z 317.676,A -85,B 0,C 180,E1 -23378.467,E2 -23378.467} C_VEL
LIN {X 0,Y 313.22,Z 318.03,A -85,B 0,C 180,E1 -23380.195,E2 -23380.195} C_VEL
LIN {X 0,Y 310.811,Z 318.33,A -85,B 0,C 180,E1 -23381.596,E2 -23381.596} C_VEL
LIN {X 0,Y 309.759,Z 318.456,A -85,B 0,C 180,E1 -23382.679,E2 -23382.679} C_VEL
LIN {X 0,Y 309.664,Z 318.466,A -85,B 0,C 180,E1 -23383.047,E2 -23383.047} C_VEL
LIN {X 0,Y 309.819,Z 318.437,A -85,B 0,C 180,E1 -23386.934,E2 -23386.934} C_VEL
LIN {X 0,Y 309.88,Z 318.423,A -85,B 0,C 180,E1 -23390.896,E2 -23390.896} C_VEL
LIN {X 0,Y 310.059,Z 318.421,A -85,B 0,C 180,E1 -23393.677,E2 -23393.677} C_VEL
LIN {X 0,Y 310.046,Z 318.406,A -85,B 0,C 180,E1 -23397.41,E2 -23397.41} C_VEL
LIN {X 0,Y 310.101,Z 318.394,A -85,B 0,C 180,E1 -23401.294,E2 -23401.294} C_VEL
LIN {X 0,Y 310.022,Z 318.422,A -85,B 0,C 180,E1 -23405.185,E2 -23405.185} C_VEL
LIN {X 0,Y 309.942,Z 318.413,A -85,B 0,C 180,E1 -23407.793,E2 -23407.793} C_VEL
LIN {X 0,Y 309.8,Z 318.434,A -85,B 0,C 180,E1 -23411.741,E2 -23411.741} C_VEL
LIN {X 0,Y 309.779,Z 318.447,A -85,B 0,C 180,E1 -23414.402,E2 -23414.402} C_VEL
LIN {X 0,Y 309.696,Z 318.449,A -85,B 0,C 180,E1 -23418.46,E2 -23418.46} C_VEL
LIN {X 0,Y 309.667,Z 318.452,A -85,B 0,C 180,E1 -23421.979,E2 -23421.979} C_VEL
LIN {X 0,Y 309.631,Z 318.467,A -85,B 0,C 180,E1 -23425.456,E2 -23425.456} C_VEL
LIN {X 0,Y 309.59,Z 318.479,A -85,B 0,C 180,E1 -23428.367,E2 -23428.367} C_VEL
LIN {X 0,Y 309.587,Z 318.472,A -85,B 0,C 180,E1 -23431.358,E2 -23431.358} C_VEL
LIN {X 0,Y 309.608,Z 318.442,A -85,B 0,C 180,E1 -23434.443,E2 -23434.443} C_VEL
LIN {X 0,Y 309.662,Z 318.447,A -85,B 0,C 180,E1 -23437.663,E2 -23437.663} C_VEL
LIN {X 0,Y 309.626,Z 318.476,A -85,B 0,C 180,E1 -23441.715,E2 -23441.715} C_VEL
LIN {X 0,Y 309.606,Z 318.646,A -85,B 0,C 180,E1 -23444.405,E2 -23444.405} C_VEL
LIN {X 0,Y 311.815,Z 325.869,A -85,B 0,C 180,E1 -23447.285,E2 -23447.285} C_VEL
LIN {X 0,Y 314.46,Z 335.15,A -85,B 0,C 180,E1 -23450.718,E2 -23450.718} C_VEL
LIN {X 0,Y 316.817,Z 344.39,A -85,B 0,C 180,E1 -23453.839,E2 -23453.839} C_VEL
LIN {X 0,Y 319.075,Z 348.799,A -85,B 0,C 180,E1 -23454.315,E2 -23454.315} C_VEL
LIN {X 0,Y 326.69,Z 364.104,A -85,B 0,C 180,E1 -23455.857,E2 -23455.857} C_VEL
LIN {X 0,Y 332.893,Z 377.762,A -85,B 0,C 180,E1 -23457.069,E2 -23457.069} C_VEL
LIN {X 0,Y 337.388,Z 405.847,A -85,B 0,C 180,E1 -23458.381,E2 -23458.381} C_VEL
LIN {X 0,Y 338.937,Z 418.541,A -85,B 0,C 180,E1 -23458.896,E2 -23458.896} C_VEL
LIN {X 0,Y 336.196,Z 484.495,A -85,B 0,C 180,E1 -23460.303,E2 -23460.303} C_VEL
LIN {X 0,Y 334.833,Z 498.801,A -85,B 0,C 180,E1 -23460.816,E2 -23460.816} C_VEL
LIN {X 0,Y 332.725,Z 513.184,A -85,B 0,C 180,E1 -23461.56,E2 -23461.56} C_VEL
LIN {X 0,Y 330.445,Z 525.101,A -85,B 0,C 180,E1 -23462.379,E2 -23462.379} C_VEL
LIN {X 0,Y 327.749,Z 537.715,A -85,B 0,C 180,E1 -23463.508,E2 -23463.508} C_VEL
LIN {X 0,Y 324.877,Z 549.221,A -85,B 0,C 180,E1 -23464.8,E2 -23464.8} C_VEL
LIN {X 0,Y 322.001,Z 559.822,A -85,B 0,C 180,E1 -23466.274,E2 -23466.274} C_VEL
LIN {X 0,Y 318.74,Z 570.362,A -85,B 0,C 180,E1 -23468.067,E2 -23468.067} C_VEL
LIN {X 0,Y 315.93,Z 579.093,A -85,B 0,C 180,E1 -23469.904,E2 -23469.904} C_VEL
LIN {X 0,Y 313.211,Z 587.51,A -85,B 0,C 180,E1 -23472.095,E2 -23472.095} C_VEL
LIN {X 0,Y 311.039,Z 594.325,A -85,B 0,C 180,E1 -23474.325,E2 -23474.325} C_VEL
LIN {X 0,Y 309.537,Z 599.051,A -85,B 0,C 180,E1 -23476.258,E2 -23476.258} C_VEL
LIN {X 0,Y 308.094,Z 604.005,A -85,B 0,C 180,E1 -23478.861,E2 -23478.861} C_VEL
LIN {X 0,Y 307.357,Z 606.75,A -85,B 0,C 180,E1 -23480.824,E2 -23480.824} C_VEL
LIN {X 0,Y 306.914,Z 609.213,A -85,B 0,C 180,E1 -23483.451,E2 -23483.451} C_VEL
LIN {X 0,Y 307.127,Z 610.551,A -85,B 0,C 180,E1 -23486.326,E2 -23486.326} C_VEL
LIN {X 0,Y 307.083,Z 615.375,A -85,B 0,C 180,E1 -23488.696,E2 -23488.696} C_VEL
LIN {X 0,Y 306.971,Z 619.094,A -85,B 0,C 180,E1 -23491.311,E2 -23491.311} C_VEL
LIN {X 0,Y 306.83,Z 621.305,A -85,B 0,C 180,E1 -23493.93,E2 -23493.93} C_VEL
LIN {X 0,Y 307.036,Z 622.117,A -85,B 0,C 180,E1 -23496.553,E2 -23496.553} C_VEL
LIN {X 0,Y 307.726,Z 621.565,A -85,B 0,C 180,E1 -23499.171,E2 -23499.171} C_VEL
LIN {X 0,Y 309.124,Z 619.659,A -85,B 0,C 180,E1 -23501.77,E2 -23501.77} C_VEL
LIN {X 0,Y 311.19,Z 616.384,A -85,B 0,C 180,E1 -23504.338,E2 -23504.338} C_VEL
LIN {X 0,Y 313.811,Z 611.654,A -85,B 0,C 180,E1 -23506.871,E2 -23506.871} C_VEL
LIN {X 0,Y 316.328,Z 607.038,A -85,B 0,C 180,E1 -23508.731,E2 -23508.731} C_VEL
LIN {X 0,Y 320.185,Z 599.436,A -85,B 0,C 180,E1 -23511.162,E2 -23511.162} C_VEL
LIN {X 0,Y 324.007,Z 591.131,A -85,B 0,C 180,E1 -23513.24,E2 -23513.24} C_VEL
LIN {X 0,Y 327.81,Z 582.602,A -85,B 0,C 180,E1 -23514.964,E2 -23514.964} C_VEL
LIN {X 0,Y 331.942,Z 572.432,A -85,B 0,C 180,E1 -23516.644,E2 -23516.644} C_VEL
LIN {X 0,Y 336.137,Z 561.323,A -85,B 0,C 180,E1 -23518.132,E2 -23518.132} C_VEL
LIN {X 0,Y 340.636,Z 547.901,A -85,B 0,C 180,E1 -23519.574,E2 -23519.574} C_VEL
LIN {X 0,Y 344.131,Z 536.029,A -85,B 0,C 180,E1 -23520.59,E2 -23520.59} C_VEL
LIN {X 0,Y 347.868,Z 521.17,A -85,B 0,C 180,E1 -23521.571,E2 -23521.571} C_VEL
LIN {X 0,Y 351.117,Z 505.497,A -85,B 0,C 180,E1 -23522.339,E2 -23522.339} C_VEL
LIN {X 0,Y 353.588,Z 487.981,A -85,B 0,C 180,E1 -23522.969,E2 -23522.969} C_VEL
LIN {X 0,Y 361.683,Z 422.793,A -85,B 0,C 180,E1 -23525.078,E2 -23525.078} C_VEL
LIN {X 0,Y 361.908,Z 406.399,A -85,B 0,C 180,E1 -23526.139,E2 -23526.139} C_VEL
LIN {X 0,Y 361.696,Z 395.291,A -85,B 0,C 180,E1 -23527.011,E2 -23527.011} C_VEL
LIN {X 0,Y 361.218,Z 393.815,A -85,B 0,C 180,E1 -23527.27,E2 -23527.27} C_VEL
LIN {X 0,Y 357.621,Z 387.701,A -85,B 0,C 180,E1 -23528.977,E2 -23528.977} C_VEL
LIN {X 0,Y 354.274,Z 382.405,A -85,B 0,C 180,E1 -23530.834,E2 -23530.834} C_VEL
LIN {X 0,Y 350.958,Z 377.637,A -85,B 0,C 180,E1 -23533.074,E2 -23533.074} C_VEL
LIN {X 0,Y 348.963,Z 375.012,A -85,B 0,C 180,E1 -23534.776,E2 -23534.776} C_VEL
LIN {X 0,Y 346.68,Z 371.907,A -85,B 0,C 180,E1 -23537.727,E2 -23537.727} C_VEL
LIN {X 0,Y 345.922,Z 371.03,A -85,B 0,C 180,E1 -23539.612,E2 -23539.612} C_VEL
LIN {X 0,Y 345.732,Z 371.398,A -85,B 0,C 180,E1 -23542.34,E2 -23542.34} C_VEL
LIN {X 0,Y 346.767,Z 373.605,A -85,B 0,C 180,E1 -23545.192,E2 -23545.192} C_VEL
LIN {X 0,Y 348.996,Z 377.372,A -85,B 0,C 180,E1 -23547.936,E2 -23547.936} C_VEL
LIN {X 0,Y 351.86,Z 382.501,A -85,B 0,C 180,E1 -23550.325,E2 -23550.325} C_VEL
LIN {X 0,Y 354.734,Z 388.045,A -85,B 0,C 180,E1 -23552.227,E2 -23552.227} C_VEL
LIN {X 0,Y 356.929,Z 392.495,A -85,B 0,C 180,E1 -23553.481,E2 -23553.481} C_VEL
LIN {X 0,Y 360.124,Z 399.541,A -85,B 0,C 180,E1 -23555.114,E2 -23555.114} C_VEL
LIN {X 0,Y 362.889,Z 406.744,A -85,B 0,C 180,E1 -23556.442,E2 -23556.442} C_VEL
LIN {X 0,Y 363.584,Z 408.648,A -85,B 0,C 180,E1 -23556.764,E2 -23556.764} C_VEL
LIN {X 0,Y 352.887,Z 492.381,A -85,B 0,C 180,E1 -23559.448,E2 -23559.448} C_VEL
LIN {X 0,Y 350.257,Z 506.97,A -85,B 0,C 180,E1 -23560.125,E2 -23560.125} C_VEL
LIN {X 0,Y 346.748,Z 522.843,A -85,B 0,C 180,E1 -23561.143,E2 -23561.143} C_VEL
LIN {X 0,Y 342.888,Z 536.836,A -85,B 0,C 180,E1 -23562.31,E2 -23562.31} C_VEL
LIN {X 0,Y 338.826,Z 549.481,A -85,B 0,C 180,E1 -23563.64,E2 -23563.64} C_VEL
LIN {X 0,Y 334.656,Z 561.007,A -85,B 0,C 180,E1 -23565.144,E2 -23565.144} C_VEL
LIN {X 0,Y 330.484,Z 571.364,A -85,B 0,C 180,E1 -23566.83,E2 -23566.83} C_VEL
LIN {X 0,Y 326.077,Z 581.335,A -85,B 0,C 180,E1 -23568.853,E2 -23568.853} C_VEL
LIN {X 0,Y 322.099,Z 589.512,A -85,B 0,C 180,E1 -23570.929,E2 -23570.929} C_VEL
LIN {X 0,Y 318.488,Z 596.153,A -85,B 0,C 180,E1 -23573.052,E2 -23573.052} C_VEL
LIN {X 0,Y 314.957,Z 602.086,A -85,B 0,C 180,E1 -23575.536,E2 -23575.536} C_VEL
LIN {X 0,Y 312.793,Z 605.451,A -85,B 0,C 180,E1 -23577.433,E2 -23577.433} C_VEL
LIN {X 0,Y 310.443,Z 608.679,A -85,B 0,C 180,E1 -23580,E2 -23580} C_VEL
LIN {X 0,Y 308.845,Z 610.466,A -85,B 0,C 180,E1 -23582.6,E2 -23582.6} C_VEL
LIN {X 0,Y 307.616,Z 610.88,A -85,B 0,C 180,E1 -23585.226,E2 -23585.226} C_VEL
LIN {X 0,Y 306.882,Z 609.898,A -85,B 0,C 180,E1 -23587.871,E2 -23587.871} C_VEL
LIN {X 0,Y 306.644,Z 607.49,A -85,B 0,C 180,E1 -23590.529,E2 -23590.529} C_VEL
LIN {X 0,Y 306.519,Z 603.541,A -85,B 0,C 180,E1 -23593.21,E2 -23593.21} C_VEL
LIN {X 0,Y 306.721,Z 599.458,A -85,B 0,C 180,E1 -23595.226,E2 -23595.226} C_VEL
LIN {X 0,Y 306.917,Z 594.286,A -85,B 0,C 180,E1 -23597.259,E2 -23597.259} C_VEL
LIN {X 0,Y 307.338,Z 586.699,A -85,B 0,C 180,E1 -23599.643,E2 -23599.643} C_VEL
LIN {X 0,Y 307.844,Z 578.603,A -85,B 0,C 180,E1 -23601.7,E2 -23601.7} C_VEL
LIN {X 0,Y 308.54,Z 568.754,A -85,B 0,C 180,E1 -23603.763,E2 -23603.763} C_VEL
LIN {X 0,Y 309.432,Z 557.732,A -85,B 0,C 180,E1 -23605.653,E2 -23605.653} C_VEL
LIN {X 0,Y 310.449,Z 545.567,A -85,B 0,C 180,E1 -23607.368,E2 -23607.368} C_VEL
LIN {X 0,Y 311.513,Z 532.041,A -85,B 0,C 180,E1 -23608.923,E2 -23608.923} C_VEL
LIN {X 0,Y 312.534,Z 518.094,A -85,B 0,C 180,E1 -23610.19,E2 -23610.19} C_VEL
LIN {X 0,Y 313.522,Z 503.755,A -85,B 0,C 180,E1 -23611.201,E2 -23611.201} C_VEL
LIN {X 0,Y 314.38,Z 488.814,A -85,B 0,C 180,E1 -23611.982,E2 -23611.982} C_VEL
LIN {X 0,Y 315.608,Z 452.392,A -85,B 0,C 180,E1 -23613.223,E2 -23613.223} C_VEL
LIN {X 0,Y 318.125,Z 385.665,A -85,B 0,C 180,E1 -23615.405,E2 -23615.405} C_VEL
LIN {X 0,Y 314.74,Z 353.332,A -85,B 0,C 180,E1 -23616.621,E2 -23616.621} C_VEL
LIN {X 0,Y 314.274,Z 345.956,A -85,B 0,C 180,E1 -23616.931,E2 -23616.931} C_VEL
LIN {X 0,Y 314.456,Z 342.562,A -85,B 0,C 180,E1 -23617.573,E2 -23617.573} C_VEL
LIN {X 0,Y 311.118,Z 325.943,A -85,B 0,C 180,E1 -23620.937,E2 -23620.937} C_VEL
LIN {X 0,Y 309.64,Z 318.476,A -85,B 0,C 180,E1 -23622.498,E2 -23622.498} C_VEL
LIN {X 0,Y 309.582,Z 318.477,A -85,B 0,C 180,E1 -23626.387,E2 -23626.387} C_VEL
LIN {X 0,Y 309.565,Z 318.479,A -85,B 0,C 180,E1 -23630.292,E2 -23630.292} C_VEL
LIN {X 0,Y 309.581,Z 318.478,A -85,B 0,C 180,E1 -23633.963,E2 -23633.963} C_VEL
LIN {X 0,Y 309.616,Z 318.468,A -85,B 0,C 180,E1 -23637.112,E2 -23637.112} C_VEL
LIN {X 0,Y 309.563,Z 318.481,A -85,B 0,C 180,E1 -23640.143,E2 -23640.143} C_VEL
LIN {X 0,Y 309.626,Z 318.469,A -85,B 0,C 180,E1 -23643.096,E2 -23643.096} C_VEL
LIN {X 0,Y 309.625,Z 318.475,A -85,B 0,C 180,E1 -23645.968,E2 -23645.968} C_VEL
LIN {X 0,Y 309.689,Z 318.466,A -85,B 0,C 180,E1 -23648.781,E2 -23648.781} C_VEL
LIN {X 0,Y 309.72,Z 318.458,A -85,B 0,C 180,E1 -23652.899,E2 -23652.899} C_VEL
LIN {X 0,Y 309.756,Z 318.485,A -85,B 0,C 180,E1 -23654.068,E2 -23654.068} C_VEL
LIN {X 0,Y 310.728,Z 321.285,A -85,B 0,C 180,E1 -23654.217,E2 -23654.217} C_VEL
LIN {X 0,Y 319.026,Z 340.272,A -85,B 0,C 180,E1 -23655.325,E2 -23655.325} C_VEL
LIN {X 0,Y 323.555,Z 353.928,A -85,B 0,C 180,E1 -23655.981,E2 -23655.981} C_VEL
LIN {X 0,Y 320.884,Z 450.372,A -85,B 0,C 180,E1 -23658.109,E2 -23658.109} C_VEL
LIN {X 0,Y 320.171,Z 464.759,A -85,B 0,C 180,E1 -23658.682,E2 -23658.682} C_VEL
LIN {X 0,Y 319.172,Z 478.58,A -85,B 0,C 180,E1 -23659.486,E2 -23659.486} C_VEL
LIN {X 0,Y 317.941,Z 491.47,A -85,B 0,C 180,E1 -23660.486,E2 -23660.486} C_VEL
LIN {X 0,Y 316.6,Z 502.591,A -85,B 0,C 180,E1 -23661.569,E2 -23661.569} C_VEL
LIN {X 0,Y 314.925,Z 514.303,A -85,B 0,C 180,E1 -23662.97,E2 -23662.97} C_VEL
LIN {X 0,Y 313.572,Z 524.955,A -85,B 0,C 180,E1 -23664.549,E2 -23664.549} C_VEL
LIN {X 0,Y 311.922,Z 535.554,A -85,B 0,C 180,E1 -23666.456,E2 -23666.456} C_VEL
LIN {X 0,Y 310.624,Z 544.295,A -85,B 0,C 180,E1 -23668.382,E2 -23668.382} C_VEL
LIN {X 0,Y 309.221,Z 552.713,A -85,B 0,C 180,E1 -23670.646,E2 -23670.646} C_VEL
LIN {X 0,Y 308.606,Z 559.528,A -85,B 0,C 180,E1 -23672.957,E2 -23672.957} C_VEL
LIN {X 0,Y 307.899,Z 564.824,A -85,B 0,C 180,E1 -23675.218,E2 -23675.218} C_VEL
LIN {X 0,Y 307.27,Z 569.477,A -85,B 0,C 180,E1 -23677.858,E2 -23677.858} C_VEL
LIN {X 0,Y 307.164,Z 572.632,A -85,B 0,C 180,E1 -23680.508,E2 -23680.508} C_VEL
LIN {X 0,Y 307.196,Z 574.426,A -85,B 0,C 180,E1 -23683.177,E2 -23683.177} C_VEL
LIN {X 0,Y 307.608,Z 574.866,A -85,B 0,C 180,E1 -23685.854,E2 -23685.854} C_VEL
LIN {X 0,Y 308.332,Z 573.949,A -85,B 0,C 180,E1 -23688.541,E2 -23688.541} C_VEL
LIN {X 0,Y 309.512,Z 571.638,A -85,B 0,C 180,E1 -23691.225,E2 -23691.225} C_VEL
LIN {X 0,Y 311.21,Z 567.856,A -85,B 0,C 180,E1 -23693.895,E2 -23693.895} C_VEL
LIN {X 0,Y 312.784,Z 563.92,A -85,B 0,C 180,E1 -23695.888,E2 -23695.888} C_VEL
LIN {X 0,Y 314.688,Z 559.018,A -85,B 0,C 180,E1 -23697.863,E2 -23697.863} C_VEL
LIN {X 0,Y 317.338,Z 551.886,A -85,B 0,C 180,E1 -23700.138,E2 -23700.138} C_VEL
LIN {X 0,Y 319.85,Z 544.351,A -85,B 0,C 180,E1 -23702.073,E2 -23702.073} C_VEL
LIN {X 0,Y 322.754,Z 535.224,A -85,B 0,C 180,E1 -23703.971,E2 -23703.971} C_VEL
LIN {X 0,Y 325.681,Z 525.082,A -85,B 0,C 180,E1 -23705.684,E2 -23705.684} C_VEL
LIN {X 0,Y 328.507,Z 513.878,A -85,B 0,C 180,E1 -23707.225,E2 -23707.225} C_VEL
LIN {X 0,Y 331.147,Z 501.879,A -85,B 0,C 180,E1 -23708.553,E2 -23708.553} C_VEL
LIN {X 0,Y 333.53,Z 488.401,A -85,B 0,C 180,E1 -23709.729,E2 -23709.729} C_VEL
LIN {X 0,Y 335.347,Z 474.88,A -85,B 0,C 180,E1 -23710.636,E2 -23710.636} C_VEL
LIN {X 0,Y 336.805,Z 460.399,A -85,B 0,C 180,E1 -23711.336,E2 -23711.336} C_VEL
LIN {X 0,Y 337.736,Z 446.401,A -85,B 0,C 180,E1 -23711.771,E2 -23711.771} C_VEL
LIN {X 0,Y 340.659,Z 374.337,A -85,B 0,C 180,E1 -23713.28,E2 -23713.28} C_VEL
LIN {X 0,Y 333.792,Z 359.606,A -85,B 0,C 180,E1 -23714.549,E2 -23714.549} C_VEL
LIN {X 0,Y 325.11,Z 343.286,A -85,B 0,C 180,E1 -23716.199,E2 -23716.199} C_VEL
LIN {X 0,Y 316.624,Z 330.068,A -85,B 0,C 180,E1 -23717.864,E2 -23717.864} C_VEL
LIN {X 0,Y 314.483,Z 326.82,A -85,B 0,C 180,E1 -23718.303,E2 -23718.303} C_VEL
LIN {X 0,Y 312.057,Z 323.063,A -85,B 0,C 180,E1 -23718.815,E2 -23718.815} C_VEL
LIN {X 0,Y 310.242,Z 320.791,A -85,B 0,C 180,E1 -23719.189,E2 -23719.189} C_VEL
LIN {X 0,Y 309.526,Z 318.486,A -85,B 0,C 180,E1 -23719.385,E2 -23719.385} C_VEL
LIN {X 0,Y 309.591,Z 318.465,A -85,B 0,C 180,E1 -23722.354,E2 -23722.354} C_VEL
LIN {X 0,Y 309.563,Z 318.453,A -85,B 0,C 180,E1 -23725.551,E2 -23725.551} C_VEL
LIN {X 0,Y 309.554,Z 318.474,A -85,B 0,C 180,E1 -23728.639,E2 -23728.639} C_VEL
LIN {X 0,Y 309.601,Z 318.468,A -85,B 0,C 180,E1 -23731.917,E2 -23731.917} C_VEL
LIN {X 0,Y 309.614,Z 318.465,A -85,B 0,C 180,E1 -23735.97,E2 -23735.97} C_VEL
LIN {X 0,Y 309.663,Z 318.47,A -85,B 0,C 180,E1 -23738.782,E2 -23738.782} C_VEL
LIN {X 0,Y 309.672,Z 318.466,A -85,B 0,C 180,E1 -23742.9,E2 -23742.9} C_VEL
LIN {X 0,Y 309.664,Z 318.466,A -85,B 0,C 180,E1 -23743.047,E2 -23743.047} C_VEL
LIN {X 0,Y 308.98,Z 318.553,A -85,B 0,C 180,E1 -23744.134,E2 -23744.134} C_VEL
LIN {X 0,Y 306.157,Z 318.9,A -85,B 0,C 180,E1 -23745.905,E2 -23745.905} C_VEL
LIN {X 0,Y 303.793,Z 319.197,A -85,B 0,C 180,E1 -23747.341,E2 -23747.341} C_VEL
LIN {X 0,Y 302.8,Z 319.325,A -85,B 0,C 180,E1 -23748.452,E2 -23748.452} C_VEL
LIN {X 0,Y 302.73,Z 319.328,A -85,B 0,C 180,E1 -23748.828,E2 -23748.828} C_VEL
LIN {X 0,Y 302.876,Z 319.301,A -85,B 0,C 180,E1 -23752.024,E2 -23752.024} C_VEL
LIN {X 0,Y 302.974,Z 319.296,A -85,B 0,C 180,E1 -23754.694,E2 -23754.694} C_VEL
LIN {X 0,Y 303.006,Z 319.282,A -85,B 0,C 180,E1 -23757.35,E2 -23757.35} C_VEL
LIN {X 0,Y 303.077,Z 319.287,A -85,B 0,C 180,E1 -23760,E2 -23760} C_VEL
LIN {X 0,Y 303.053,Z 319.291,A -85,B 0,C 180,E1 -23763.976,E2 -23763.976} C_VEL
LIN {X 0,Y 302.967,Z 319.284,A -85,B 0,C 180,E1 -23766.638,E2 -23766.638} C_VEL
LIN {X 0,Y 302.774,Z 319.321,A -85,B 0,C 180,E1 -23770.665,E2 -23770.665} C_VEL
LIN {X 0,Y 302.793,Z 319.31,A -85,B 0,C 180,E1 -23773.711,E2 -23773.711} C_VEL
LIN {X 0,Y 302.654,Z 319.325,A -85,B 0,C 180,E1 -23778.412,E2 -23778.412} C_VEL
LIN {X 0,Y 302.6,Z 319.332,A -85,B 0,C 180,E1 -23782.206,E2 -23782.206} C_VEL
LIN {X 0,Y 302.56,Z 319.342,A -85,B 0,C 180,E1 -23786.095,E2 -23786.095} C_VEL
LIN {X 0,Y 302.514,Z 319.359,A -85,B 0,C 180,E1 -23789.094,E2 -23789.094} C_VEL
LIN {X 0,Y 302.555,Z 319.355,A -85,B 0,C 180,E1 -23792.173,E2 -23792.173} C_VEL
LIN {X 0,Y 302.61,Z 319.303,A -85,B 0,C 180,E1 -23795.898,E2 -23795.898} C_VEL
LIN {X 0,Y 302.579,Z 319.352,A -85,B 0,C 180,E1 -23798.684,E2 -23798.684} C_VEL
LIN {X 0,Y 302.562,Z 319.351,A -85,B 0,C 180,E1 -23802.205,E2 -23802.205} C_VEL
LIN {X 0,Y 302.565,Z 319.528,A -85,B 0,C 180,E1 -23803.3,E2 -23803.3} C_VEL
LIN {X 0,Y 304.862,Z 327.002,A -85,B 0,C 180,E1 -23806.433,E2 -23806.433} C_VEL
LIN {X 0,Y 307.274,Z 335.434,A -85,B 0,C 180,E1 -23809.668,E2 -23809.668} C_VEL
LIN {X 0,Y 309.551,Z 343.945,A -85,B 0,C 180,E1 -23812.66,E2 -23812.66} C_VEL
LIN {X 0,Y 311.845,Z 348.318,A -85,B 0,C 180,E1 -23813.169,E2 -23813.169} C_VEL
LIN {X 0,Y 317.922,Z 360.038,A -85,B 0,C 180,E1 -23814.468,E2 -23814.468} C_VEL
LIN {X 0,Y 325.28,Z 375.635,A -85,B 0,C 180,E1 -23815.98,E2 -23815.98} C_VEL
LIN {X 0,Y 327.61,Z 381.325,A -85,B 0,C 180,E1 -23816.459,E2 -23816.459} C_VEL
LIN {X 0,Y 331.704,Z 407.609,A -85,B 0,C 180,E1 -23817.712,E2 -23817.712} C_VEL
LIN {X 0,Y 333.16,Z 419.622,A -85,B 0,C 180,E1 -23818.216,E2 -23818.216} C_VEL
LIN {X 0,Y 330.349,Z 483.673,A -85,B 0,C 180,E1 -23819.591,E2 -23819.591} C_VEL
LIN {X 0,Y 328.983,Z 498.101,A -85,B 0,C 180,E1 -23820.113,E2 -23820.113} C_VEL
LIN {X 0,Y 326.903,Z 511.998,A -85,B 0,C 180,E1 -23820.83,E2 -23820.83} C_VEL
LIN {X 0,Y 324.203,Z 525.834,A -85,B 0,C 180,E1 -23821.8,E2 -23821.8} C_VEL
LIN {X 0,Y 321.436,Z 538.226,A -85,B 0,C 180,E1 -23822.946,E2 -23822.946} C_VEL
LIN {X 0,Y 318.419,Z 549.813,A -85,B 0,C 180,E1 -23824.288,E2 -23824.288} C_VEL
LIN {X 0,Y 315.535,Z 560.041,A -85,B 0,C 180,E1 -23825.757,E2 -23825.757} C_VEL
LIN {X 0,Y 312.165,Z 570.476,A -85,B 0,C 180,E1 -23827.58,E2 -23827.58} C_VEL
LIN {X 0,Y 308.821,Z 580.422,A -85,B 0,C 180,E1 -23829.768,E2 -23829.768} C_VEL
LIN {X 0,Y 306.078,Z 588.482,A -85,B 0,C 180,E1 -23832.008,E2 -23832.008} C_VEL
LIN {X 0,Y 304.193,Z 594.198,A -85,B 0,C 180,E1 -23833.963,E2 -23833.963} C_VEL
LIN {X 0,Y 302.163,Z 600.24,A -85,B 0,C 180,E1 -23836.6,E2 -23836.6} C_VEL
LIN {X 0,Y 300.777,Z 604.739,A -85,B 0,C 180,E1 -23839.266,E2 -23839.266} C_VEL
LIN {X 0,Y 299.975,Z 607.821,A -85,B 0,C 180,E1 -23841.95,E2 -23841.95} C_VEL
LIN {X 0,Y 299.863,Z 609.575,A -85,B 0,C 180,E1 -23844.642,E2 -23844.642} C_VEL
LIN {X 0,Y 300.066,Z 610.121,A -85,B 0,C 180,E1 -23846.49,E2 -23846.49} C_VEL
LIN {X 0,Y 300.033,Z 614.569,A -85,B 0,C 180,E1 -23848.666,E2 -23848.666} C_VEL
LIN {X 0,Y 299.959,Z 616.745,A -85,B 0,C 180,E1 -23850.003,E2 -23850.003} C_VEL
LIN {X 0,Y 299.909,Z 618.512,A -85,B 0,C 180,E1 -23851.342,E2 -23851.342} C_VEL
LIN {X 0,Y 299.769,Z 620.908,A -85,B 0,C 180,E1 -23854.023,E2 -23854.023} C_VEL
LIN {X 0,Y 299.955,Z 621.907,A -85,B 0,C 180,E1 -23856.708,E2 -23856.708} C_VEL
LIN {X 0,Y 300.706,Z 621.552,A -85,B 0,C 180,E1 -23859.387,E2 -23859.387} C_VEL
LIN {X 0,Y 302.17,Z 619.858,A -85,B 0,C 180,E1 -23862.045,E2 -23862.045} C_VEL
LIN {X 0,Y 304.305,Z 616.799,A -85,B 0,C 180,E1 -23864.67,E2 -23864.67} C_VEL
LIN {X 0,Y 307.05,Z 612.317,A -85,B 0,C 180,E1 -23867.254,E2 -23867.254} C_VEL
LIN {X 0,Y 310.656,Z 606.296,A -85,B 0,C 180,E1 -23869.771,E2 -23869.771} C_VEL
LIN {X 0,Y 314.21,Z 599.624,A -85,B 0,C 180,E1 -23871.928,E2 -23871.928} C_VEL
LIN {X 0,Y 318.264,Z 591.466,A -85,B 0,C 180,E1 -23874.029,E2 -23874.029} C_VEL
LIN {X 0,Y 323.012,Z 581.455,A -85,B 0,C 180,E1 -23876.05,E2 -23876.05} C_VEL
LIN {X 0,Y 327.333,Z 571.186,A -85,B 0,C 180,E1 -23877.74,E2 -23877.74} C_VEL
LIN {X 0,Y 332.227,Z 558.812,A -85,B 0,C 180,E1 -23879.356,E2 -23879.356} C_VEL
LIN {X 0,Y 336.511,Z 546.243,A -85,B 0,C 180,E1 -23880.664,E2 -23880.664} C_VEL
LIN {X 0,Y 340.23,Z 534.093,A -85,B 0,C 180,E1 -23881.67,E2 -23881.67} C_VEL
LIN {X 0,Y 343.874,Z 520.017,A -85,B 0,C 180,E1 -23882.585,E2 -23882.585} C_VEL
LIN {X 0,Y 347.125,Z 504.786,A -85,B 0,C 180,E1 -23883.317,E2 -23883.317} C_VEL
LIN {X 0,Y 349.775,Z 486.523,A -85,B 0,C 180,E1 -23883.978,E2 -23883.978} C_VEL
LIN {X 0,Y 357.932,Z 423.913,A -85,B 0,C 180,E1 -23886.03,E2 -23886.03} C_VEL
LIN {X 0,Y 358.299,Z 408.519,A -85,B 0,C 180,E1 -23887.056,E2 -23887.056} C_VEL
LIN {X 0,Y 358.219,Z 399.407,A -85,B 0,C 180,E1 -23887.791,E2 -23887.791} C_VEL
LIN {X 0,Y 354.891,Z 393.479,A -85,B 0,C 180,E1 -23889.497,E2 -23889.497} C_VEL
LIN {X 0,Y 351.915,Z 388.655,A -85,B 0,C 180,E1 -23891.238,E2 -23891.238} C_VEL
LIN {X 0,Y 348.899,Z 384.126,A -85,B 0,C 180,E1 -23893.41,E2 -23893.41} C_VEL
LIN {X 0,Y 346.961,Z 381.554,A -85,B 0,C 180,E1 -23895.176,E2 -23895.176} C_VEL
LIN {X 0,Y 345.004,Z 378.732,A -85,B 0,C 180,E1 -23897.934,E2 -23897.934} C_VEL
LIN {X 0,Y 344.429,Z 378.002,A -85,B 0,C 180,E1 -23899.401,E2 -23899.401} C_VEL
LIN {X 0,Y 344.116,Z 378.088,A -85,B 0,C 180,E1 -23901.579,E2 -23901.579} C_VEL
LIN {X 0,Y 344.639,Z 379.576,A -85,B 0,C 180,E1 -23904.091,E2 -23904.091} C_VEL
LIN {X 0,Y 345.892,Z 382.022,A -85,B 0,C 180,E1 -23906.292,E2 -23906.292} C_VEL
LIN {X 0,Y 347.319,Z 384.449,A -85,B 0,C 180,E1 -23907.893,E2 -23907.893} C_VEL
LIN {X 0,Y 349.78,Z 389.102,A -85,B 0,C 180,E1 -23910.045,E2 -23910.045} C_VEL
LIN {X 0,Y 352.304,Z 394.167,A -85,B 0,C 180,E1 -23911.806,E2 -23911.806} C_VEL
LIN {X 0,Y 354.672,Z 399.281,A -85,B 0,C 180,E1 -23913.244,E2 -23913.244} C_VEL
LIN {X 0,Y 357.971,Z 407.147,A -85,B 0,C 180,E1 -23915.022,E2 -23915.022} C_VEL
LIN {X 0,Y 359.587,Z 412.167,A -85,B 0,C 180,E1 -23915.891,E2 -23915.891} C_VEL
LIN {X 0,Y 348.81,Z 492.731,A -85,B 0,C 180,E1 -23918.501,E2 -23918.501} C_VEL
LIN {X 0,Y 345.938,Z 507.803,A -85,B 0,C 180,E1 -23919.21,E2 -23919.21} C_VEL
LIN {X 0,Y 342.554,Z 522.48,A -85,B 0,C 180,E1 -23920.157,E2 -23920.157} C_VEL
LIN {X 0,Y 338.601,Z 536.273,A -85,B 0,C 180,E1 -23921.298,E2 -23921.298} C_VEL
LIN {X 0,Y 334.332,Z 549.02,A -85,B 0,C 180,E1 -23922.63,E2 -23922.63} C_VEL
LIN {X 0,Y 330.342,Z 559.615,A -85,B 0,C 180,E1 -23923.999,E2 -23923.999} C_VEL
LIN {X 0,Y 325.948,Z 570.115,A -85,B 0,C 180,E1 -23925.659,E2 -23925.659} C_VEL
LIN {X 0,Y 321.805,Z 579.156,A -85,B 0,C 180,E1 -23927.428,E2 -23927.428} C_VEL
LIN {X 0,Y 317.477,Z 587.725,A -85,B 0,C 180,E1 -23929.513,E2 -23929.513} C_VEL
LIN {X 0,Y 313.54,Z 594.711,A -85,B 0,C 180,E1 -23931.651,E2 -23931.651} C_VEL
LIN {X 0,Y 309.979,Z 600.409,A -85,B 0,C 180,E1 -23933.872,E2 -23933.872} C_VEL
LIN {X 0,Y 307.136,Z 604.669,A -85,B 0,C 180,E1 -23936.077,E2 -23936.077} C_VEL
LIN {X 0,Y 304.394,Z 608.209,A -85,B 0,C 180,E1 -23938.681,E2 -23938.681} C_VEL
LIN {X 0,Y 302.417,Z 610.323,A -85,B 0,C 180,E1 -23941.327,E2 -23941.327} C_VEL
LIN {X 0,Y 301.039,Z 611.075,A -85,B 0,C 180,E1 -23944.003,E2 -23944.003} C_VEL
LIN {X 0,Y 300.047,Z 610.457,A -85,B 0,C 180,E1 -23946.703,E2 -23946.703} C_VEL
LIN {X 0,Y 299.584,Z 608.438,A -85,B 0,C 180,E1 -23949.42,E2 -23949.42} C_VEL
LIN {X 0,Y 299.554,Z 606.778,A -85,B 0,C 180,E1 -23950.85,E2 -23950.85} C_VEL
LIN {X 0,Y 299.475,Z 602.499,A -85,B 0,C 180,E1 -23953.526,E2 -23953.526} C_VEL
LIN {X 0,Y 299.709,Z 598.138,A -85,B 0,C 180,E1 -23955.591,E2 -23955.591} C_VEL
LIN {X 0,Y 299.952,Z 591.53,A -85,B 0,C 180,E1 -23958.024,E2 -23958.024} C_VEL
LIN {X 0,Y 300.371,Z 584.489,A -85,B 0,C 180,E1 -23960.118,E2 -23960.118} C_VEL
LIN {X 0,Y 300.94,Z 575.89,A -85,B 0,C 180,E1 -23962.224,E2 -23962.224} C_VEL
LIN {X 0,Y 301.704,Z 565.408,A -85,B 0,C 180,E1 -23964.336,E2 -23964.336} C_VEL
LIN {X 0,Y 302.533,Z 554.829,A -85,B 0,C 180,E1 -23966.097,E2 -23966.097} C_VEL
LIN {X 0,Y 303.517,Z 543.432,A -85,B 0,C 180,E1 -23967.674,E2 -23967.674} C_VEL
LIN {X 0,Y 304.57,Z 530.001,A -85,B 0,C 180,E1 -23969.185,E2 -23969.185} C_VEL
LIN {X 0,Y 305.523,Z 516.728,A -85,B 0,C 180,E1 -23970.385,E2 -23970.385} C_VEL
LIN {X 0,Y 306.537,Z 502.083,A -85,B 0,C 180,E1 -23971.417,E2 -23971.417} C_VEL
LIN {X 0,Y 307.385,Z 487.314,A -85,B 0,C 180,E1 -23972.172,E2 -23972.172} C_VEL
LIN {X 0,Y 311.199,Z 386.774,A -85,B 0,C 180,E1 -23975.597,E2 -23975.597} C_VEL
LIN {X 0,Y 307.848,Z 354.46,A -85,B 0,C 180,E1 -23976.845,E2 -23976.845} C_VEL
LIN {X 0,Y 307.311,Z 346.218,A -85,B 0,C 180,E1 -23977.175,E2 -23977.175} C_VEL
LIN {X 0,Y 307.44,Z 343.484,A -85,B 0,C 180,E1 -23977.701,E2 -23977.701} C_VEL
LIN {X 0,Y 303.943,Z 326.212,A -85,B 0,C 180,E1 -23981.246,E2 -23981.246} C_VEL
LIN {X 0,Y 302.579,Z 319.355,A -85,B 0,C 180,E1 -23982.684,E2 -23982.684} C_VEL
LIN {X 0,Y 302.525,Z 319.353,A -85,B 0,C 180,E1 -23986.001,E2 -23986.001} C_VEL
LIN {X 0,Y 302.505,Z 319.359,A -85,B 0,C 180,E1 -23989.828,E2 -23989.828} C_VEL
LIN {X 0,Y 302.559,Z 319.35,A -85,B 0,C 180,E1 -23994.123,E2 -23994.123} C_VEL
LIN {X 0,Y 302.518,Z 319.354,A -85,B 0,C 180,E1 -23997.82,E2 -23997.82} C_VEL
LIN {X 0,Y 302.57,Z 319.345,A -85,B 0,C 180,E1 -24001.605,E2 -24001.605} C_VEL
LIN {X 0,Y 302.562,Z 319.353,A -85,B 0,C 180,E1 -24005.37,E2 -24005.37} C_VEL
LIN {X 0,Y 302.655,Z 319.344,A -85,B 0,C 180,E1 -24008.263,E2 -24008.263} C_VEL
LIN {X 0,Y 302.68,Z 319.335,A -85,B 0,C 180,E1 -24012.489,E2 -24012.489} C_VEL
LIN {X 0,Y 302.695,Z 319.335,A -85,B 0,C 180,E1 -24013.487,E2 -24013.487} C_VEL
LIN {X 0,Y 303.806,Z 322.361,A -85,B 0,C 180,E1 -24013.675,E2 -24013.675} C_VEL
LIN {X 0,Y 312.827,Z 342.895,A -85,B 0,C 180,E1 -24014.918,E2 -24014.918} C_VEL
LIN {X 0,Y 316.961,Z 355.562,A -85,B 0,C 180,E1 -24015.541,E2 -24015.541} C_VEL
LIN {X 0,Y 314.191,Z 450.998,A -85,B 0,C 180,E1 -24017.688,E2 -24017.688} C_VEL
LIN {X 0,Y 313.471,Z 465.304,A -85,B 0,C 180,E1 -24018.273,E2 -24018.273} C_VEL
LIN {X 0,Y 312.437,Z 479.091,A -85,B 0,C 180,E1 -24019.093,E2 -24019.093} C_VEL
LIN {X 0,Y 311.179,Z 491.955,A -85,B 0,C 180,E1 -24020.114,E2 -24020.114} C_VEL
LIN {X 0,Y 309.789,Z 503.065,A -85,B 0,C 180,E1 -24021.218,E2 -24021.218} C_VEL
LIN {X 0,Y 308.071,Z 514.765,A -85,B 0,C 180,E1 -24022.649,E2 -24022.649} C_VEL
LIN {X 0,Y 306.55,Z 526.374,A -85,B 0,C 180,E1 -24024.424,E2 -24024.424} C_VEL
LIN {X 0,Y 304.848,Z 536.812,A -85,B 0,C 180,E1 -24026.374,E2 -24026.374} C_VEL
LIN {X 0,Y 303.534,Z 545.411,A -85,B 0,C 180,E1 -24028.344,E2 -24028.344} C_VEL
LIN {X 0,Y 302.132,Z 553.691,A -85,B 0,C 180,E1 -24030.661,E2 -24030.661} C_VEL
LIN {X 0,Y 301.553,Z 559.828,A -85,B 0,C 180,E1 -24032.809,E2 -24032.809} C_VEL
LIN {X 0,Y 300.771,Z 565.591,A -85,B 0,C 180,E1 -24035.342,E2 -24035.342} C_VEL
LIN {X 0,Y 300.155,Z 570.128,A -85,B 0,C 180,E1 -24038.045,E2 -24038.045} C_VEL
LIN {X 0,Y 300.081,Z 573.198,A -85,B 0,C 180,E1 -24040.759,E2 -24040.759} C_VEL
LIN {X 0,Y 300.129,Z 574.911,A -85,B 0,C 180,E1 -24043.493,E2 -24043.493} C_VEL
LIN {X 0,Y 300.591,Z 575.267,A -85,B 0,C 180,E1 -24046.234,E2 -24046.234} C_VEL
LIN {X 0,Y 301.398,Z 574.266,A -85,B 0,C 180,E1 -24048.983,E2 -24048.983} C_VEL
LIN {X 0,Y 302.689,Z 571.868,A -85,B 0,C 180,E1 -24051.727,E2 -24051.727} C_VEL
LIN {X 0,Y 304.516,Z 567.967,A -85,B 0,C 180,E1 -24054.455,E2 -24054.455} C_VEL
LIN {X 0,Y 306.818,Z 562.403,A -85,B 0,C 180,E1 -24057.163,E2 -24057.163} C_VEL
LIN {X 0,Y 309.373,Z 556.049,A -85,B 0,C 180,E1 -24059.497,E2 -24059.497} C_VEL
LIN {X 0,Y 312.267,Z 548.036,A -85,B 0,C 180,E1 -24061.814,E2 -24061.814} C_VEL
LIN {X 0,Y 315.132,Z 539.632,A -85,B 0,C 180,E1 -24063.753,E2 -24063.753} C_VEL
LIN {X 0,Y 318.431,Z 529.069,A -85,B 0,C 180,E1 -24065.721,E2 -24065.721} C_VEL
LIN {X 0,Y 321.48,Z 517.848,A -85,B 0,C 180,E1 -24067.393,E2 -24067.393} C_VEL
LIN {X 0,Y 324.258,Z 506.242,A -85,B 0,C 180,E1 -24068.784,E2 -24068.784} C_VEL
LIN {X 0,Y 326.51,Z 495.117,A -85,B 0,C 180,E1 -24069.868,E2 -24069.868} C_VEL
LIN {X 0,Y 328.525,Z 482.412,A -85,B 0,C 180,E1 -24070.861,E2 -24070.861} C_VEL
LIN {X 0,Y 330.152,Z 469.432,A -85,B 0,C 180,E1 -24071.63,E2 -24071.63} C_VEL
LIN {X 0,Y 331.372,Z 455.997,A -85,B 0,C 180,E1 -24072.197,E2 -24072.197} C_VEL
LIN {X 0,Y 332.23,Z 438.749,A -85,B 0,C 180,E1 -24072.646,E2 -24072.646} C_VEL
LIN {X 0,Y 334.84,Z 376.453,A -85,B 0,C 180,E1 -24073.962,E2 -24073.962} C_VEL
LIN {X 0,Y 327.868,Z 361.561,A -85,B 0,C 180,E1 -24075.299,E2 -24075.299} C_VEL
LIN {X 0,Y 319.893,Z 346.707,A -85,B 0,C 180,E1 -24076.871,E2 -24076.871} C_VEL
LIN {X 0,Y 310.669,Z 332.287,A -85,B 0,C 180,E1 -24078.763,E2 -24078.763} C_VEL
LIN {X 0,Y 307.431,Z 327.662,A -85,B 0,C 180,E1 -24079.455,E2 -24079.455} C_VEL
LIN {X 0,Y 304.928,Z 323.849,A -85,B 0,C 180,E1 -24080.014,E2 -24080.014} C_VEL
LIN {X 0,Y 303.194,Z 321.615,A -85,B 0,C 180,E1 -24080.397,E2 -24080.397} C_VEL
LIN {X 0,Y 302.509,Z 319.356,A -85,B 0,C 180,E1 -24080.611,E2 -24080.611} C_VEL
LIN {X 0,Y 302.525,Z 319.321,A -85,B 0,C 180,E1 -24084.632,E2 -24084.632} C_VEL
LIN {X 0,Y 302.514,Z 319.359,A -85,B 0,C 180,E1 -24087.823,E2 -24087.823} C_VEL
LIN {X 0,Y 302.56,Z 319.349,A -85,B 0,C 180,E1 -24091.6,E2 -24091.6} C_VEL
LIN {X 0,Y 302.565,Z 319.349,A -85,B 0,C 180,E1 -24095.373,E2 -24095.373} C_VEL
LIN {X 0,Y 302.629,Z 319.344,A -85,B 0,C 180,E1 -24098.264,E2 -24098.264} C_VEL
LIN {X 0,Y 302.636,Z 319.339,A -85,B 0,C 180,E1 -24102.489,E2 -24102.489} C_VEL
LIN {X 0,Y 302.767,Z 319.312,A -85,B 0,C 180,E1 -24106.624,E2 -24106.624} C_VEL
LIN {X 0,Y 302.73,Z 319.328,A -85,B 0,C 180,E1 -24108.828,E2 -24108.828} C_VEL
LIN {X 0,Y 302.107,Z 319.407,A -85,B 0,C 180,E1 -24109.939,E2 -24109.939} C_VEL
LIN {X 0,Y 299.343,Z 319.761,A -85,B 0,C 180,E1 -24111.75,E2 -24111.75} C_VEL
LIN {X 0,Y 296.995,Z 320.055,A -85,B 0,C 180,E1 -24113.22,E2 -24113.22} C_VEL
LIN {X 0,Y 296.003,Z 320.17,A -85,B 0,C 180,E1 -24114.356,E2 -24114.356} C_VEL
LIN {X 0,Y 295.931,Z 320.172,A -85,B 0,C 180,E1 -24114.741,E2 -24114.741} C_VEL
LIN {X 0,Y 296.057,Z 320.163,A -85,B 0,C 180,E1 -24118.644,E2 -24118.644} C_VEL
LIN {X 0,Y 296.057,Z 320.143,A -85,B 0,C 180,E1 -24121.356,E2 -24121.356} C_VEL
LIN {X 0,Y 296.023,Z 320.167,A -85,B 0,C 180,E1 -24124.071,E2 -24124.071} C_VEL
LIN {X 0,Y 295.914,Z 320.161,A -85,B 0,C 180,E1 -24126.797,E2 -24126.797} C_VEL
LIN {X 0,Y 295.733,Z 320.195,A -85,B 0,C 180,E1 -24130.922,E2 -24130.922} C_VEL
LIN {X 0,Y 295.748,Z 320.188,A -85,B 0,C 180,E1 -24133.841,E2 -24133.841} C_VEL
LIN {X 0,Y 295.62,Z 320.203,A -85,B 0,C 180,E1 -24138.614,E2 -24138.614} C_VEL
LIN {X 0,Y 295.563,Z 320.208,A -85,B 0,C 180,E1 -24142.456,E2 -24142.456} C_VEL
LIN {X 0,Y 295.534,Z 320.219,A -85,B 0,C 180,E1 -24145.767,E2 -24145.767} C_VEL
LIN {X 0,Y 295.49,Z 320.226,A -85,B 0,C 180,E1 -24149.854,E2 -24149.854} C_VEL
LIN {X 0,Y 295.49,Z 320.207,A -85,B 0,C 180,E1 -24153.944,E2 -24153.944} C_VEL
LIN {X 0,Y 295.542,Z 320.185,A -85,B 0,C 180,E1 -24156.335,E2 -24156.335} C_VEL
LIN {X 0,Y 295.521,Z 320.225,A -85,B 0,C 180,E1 -24159.788,E2 -24159.788} C_VEL
LIN {X 0,Y 295.531,Z 320.274,A -85,B 0,C 180,E1 -24162.065,E2 -24162.065} C_VEL
LIN {X 0,Y 298.412,Z 329.756,A -85,B 0,C 180,E1 -24166.201,E2 -24166.201} C_VEL
